LIN {X 0,Y 298.481,Z 502.932,A -85,B 0,C 180,E1 -16460.513,E2 -16460.513} C_VEL
LIN {X 0,Y 297.98,Z 506.123,A -85,B 0,C 180,E1 -16462.135,E2 -16462.135} C_VEL
LIN {X 0,Y 297.332,Z 509.748,A -85,B 0,C 180,E1 -16464.575,E2 -16464.575} C_VEL
LIN {X 0,Y 297.148,Z 511.131,A -85,B 0,C 180,E1 -16465.931,E2 -16465.931} C_VEL
LIN {X 0,Y 297.066,Z 512.111,A -85,B 0,C 180,E1 -16467.288,E2 -16467.288} C_VEL
LIN {X 0,Y 296.924,Z 512.947,A -85,B 0,C 180,E1 -16470,E2 -16470} C_VEL
LIN {X 0,Y 297.047,Z 512.175,A -85,B 0,C 180,E1 -16472.712,E2 -16472.712} C_VEL
LIN {X 0,Y 297.329,Z 509.873,A -85,B 0,C 180,E1 -16475.426,E2 -16475.426} C_VEL
LIN {X 0,Y 297.887,Z 506.563,A -85,B 0,C 180,E1 -16477.733,E2 -16477.733} C_VEL
LIN {X 0,Y 298.7,Z 501.616,A -85,B 0,C 180,E1 -16480.164,E2 -16480.164} C_VEL
LIN {X 0,Y 299.966,Z 495.208,A -85,B 0,C 180,E1 -16482.517,E2 -16482.517} C_VEL
LIN {X 0,Y 301.198,Z 488.167,A -85,B 0,C 180,E1 -16484.527,E2 -16484.527} C_VEL
LIN {X 0,Y 302.803,Z 479.382,A -85,B 0,C 180,E1 -16486.518,E2 -16486.518} C_VEL
LIN {X 0,Y 304.304,Z 470.362,A -85,B 0,C 180,E1 -16488.167,E2 -16488.167} C_VEL
LIN {X 0,Y 305.67,Z 460.096,A -85,B 0,C 180,E1 -16489.687,E2 -16489.687} C_VEL
LIN {X 0,Y 307.036,Z 449.246,A -85,B 0,C 180,E1 -16490.956,E2 -16490.956} C_VEL
LIN {X 0,Y 307.418,Z 446.051,A -85,B 0,C 180,E1 -16491.28,E2 -16491.28} C_VEL
LIN {X 0,Y 305.864,Z 437.325,A -85,B 0,C 180,E1 -16492.242,E2 -16492.242} C_VEL
LIN {X 0,Y 302.839,Z 425.594,A -85,B 0,C 180,E1 -16493.382,E2 -16493.382} C_VEL
LIN {X 0,Y 298.696,Z 412.913,A -85,B 0,C 180,E1 -16494.408,E2 -16494.408} C_VEL
LIN {X 0,Y 297.744,Z 409.886,A -85,B 0,C 180,E1 -16494.623,E2 -16494.623} C_VEL
LIN {X 0,Y 297.824,Z 406.969,A -85,B 0,C 180,E1 -16498.162,E2 -16498.162} C_VEL
LIN {X 0,Y 297.994,Z 404.067,A -85,B 0,C 180,E1 -16501.892,E2 -16501.892} C_VEL
LIN {X 0,Y 298.002,Z 403.367,A -85,B 0,C 180,E1 -16502.849,E2 -16502.849} C_VEL
LIN {X 0,Y 298.372,Z 403.32,A -85,B 0,C 180,E1 -16506.788,E2 -16506.788} C_VEL
LIN {X 0,Y 298.401,Z 403.313,A -85,B 0,C 180,E1 -16509.488,E2 -16509.488} C_VEL
LIN {X 0,Y 298.401,Z 403.313,A -85,B 0,C 180,E1 -16513.103,E2 -16513.103} C_VEL
LIN {X 0,Y 298.405,Z 403.313,A -85,B 0,C 180,E1 -16516.921,E2 -16516.921} C_VEL
LIN {X 0,Y 298.418,Z 403.309,A -85,B 0,C 180,E1 -16521.004,E2 -16521.004} C_VEL
LIN {X 0,Y 298.436,Z 403.311,A -85,B 0,C 180,E1 -16523.932,E2 -16523.932} C_VEL
LIN {X 0,Y 298.398,Z 403.316,A -85,B 0,C 180,E1 -16527.984,E2 -16527.984} C_VEL
LIN {X 0,Y 298.462,Z 403.308,A -85,B 0,C 180,E1 -16531.904,E2 -16531.904} C_VEL
LIN {X 0,Y 298.487,Z 403.301,A -85,B 0,C 180,E1 -16534.924,E2 -16534.924} C_VEL
LIN {X 0,Y 298.444,Z 403.308,A -85,B 0,C 180,E1 -16539.315,E2 -16539.315} C_VEL
LIN {X 0,Y 298.541,Z 403.298,A -85,B 0,C 180,E1 -16542.179,E2 -16542.179} C_VEL
LIN {X 0,Y 298.597,Z 403.288,A -85,B 0,C 180,E1 -16544.995,E2 -16544.995} C_VEL
LIN {X 0,Y 298.595,Z 403.288,A -85,B 0,C 180,E1 -16549.147,E2 -16549.147} C_VEL
LIN {X 0,Y 298.659,Z 403.281,A -85,B 0,C 180,E1 -16550.741,E2 -16550.741} C_VEL
LIN {X 0,Y 298.057,Z 403.359,A -85,B 0,C 180,E1 -16551.868,E2 -16551.868} C_VEL
LIN {X 0,Y 295.127,Z 403.725,A -85,B 0,C 180,E1 -16553.699,E2 -16553.699} C_VEL
LIN {X 0,Y 292.661,Z 404.03,A -85,B 0,C 180,E1 -16555.186,E2 -16555.186} C_VEL
LIN {X 0,Y 291.704,Z 404.15,A -85,B 0,C 180,E1 -16556.341,E2 -16556.341} C_VEL
LIN {X 0,Y 291.685,Z 404.15,A -85,B 0,C 180,E1 -16556.731,E2 -16556.731} C_VEL
LIN {X 0,Y 291.969,Z 404.118,A -85,B 0,C 180,E1 -16560,E2 -16560} C_VEL
LIN {X 0,Y 291.793,Z 404.138,A -85,B 0,C 180,E1 -16562.761,E2 -16562.761} C_VEL
LIN {X 0,Y 291.751,Z 404.142,A -85,B 0,C 180,E1 -16566.918,E2 -16566.918} C_VEL
LIN {X 0,Y 291.634,Z 404.16,A -85,B 0,C 180,E1 -16569.712,E2 -16569.712} C_VEL
LIN {X 0,Y 291.527,Z 404.17,A -85,B 0,C 180,E1 -16573.95,E2 -16573.95} C_VEL
LIN {X 0,Y 291.491,Z 404.173,A -85,B 0,C 180,E1 -16576.818,E2 -16576.818} C_VEL
LIN {X 0,Y 291.454,Z 404.179,A -85,B 0,C 180,E1 -16579.875,E2 -16579.875} C_VEL
LIN {X 0,Y 291.404,Z 404.185,A -85,B 0,C 180,E1 -16584.205,E2 -16584.205} C_VEL
LIN {X 0,Y 291.423,Z 404.186,A -85,B 0,C 180,E1 -16587.272,E2 -16587.272} C_VEL
LIN {X 0,Y 291.337,Z 404.195,A -85,B 0,C 180,E1 -16590.437,E2 -16590.437} C_VEL
LIN {X 0,Y 291.348,Z 404.195,A -85,B 0,C 180,E1 -16593.698,E2 -16593.698} C_VEL
LIN {X 0,Y 291.379,Z 404.189,A -85,B 0,C 180,E1 -16597.254,E2 -16597.254} C_VEL
LIN {X 0,Y 291.384,Z 404.329,A -85,B 0,C 180,E1 -16598.622,E2 -16598.622} C_VEL
LIN {X 0,Y 292.173,Z 408.492,A -85,B 0,C 180,E1 -16602.339,E2 -16602.339} C_VEL
LIN {X 0,Y 292.99,Z 412.972,A -85,B 0,C 180,E1 -16606.023,E2 -16606.023} C_VEL
LIN {X 0,Y 293.883,Z 418.089,A -85,B 0,C 180,E1 -16609.93,E2 -16609.93} C_VEL
LIN {X 0,Y 294.289,Z 420.975,A -85,B 0,C 180,E1 -16612.007,E2 -16612.007} C_VEL
LIN {X 0,Y 294.149,Z 424.38,A -85,B 0,C 180,E1 -16614.326,E2 -16614.326} C_VEL
LIN {X 0,Y 293.105,Z 430.281,A -85,B 0,C 180,E1 -16618.162,E2 -16618.162} C_VEL
LIN {X 0,Y 292.109,Z 436.327,A -85,B 0,C 180,E1 -16622.02,E2 -16622.02} C_VEL
LIN {X 0,Y 291.475,Z 440.717,A -85,B 0,C 180,E1 -16624.804,E2 -16624.804} C_VEL
LIN {X 0,Y 294.39,Z 454.459,A -85,B 0,C 180,E1 -16625.683,E2 -16625.683} C_VEL
LIN {X 0,Y 296.244,Z 466.513,A -85,B 0,C 180,E1 -16626.656,E2 -16626.656} C_VEL
LIN {X 0,Y 297.356,Z 478.025,A -85,B 0,C 180,E1 -16627.78,E2 -16627.78} C_VEL
LIN {X 0,Y 297.893,Z 489.194,A -85,B 0,C 180,E1 -16629.094,E2 -16629.094} C_VEL
LIN {X 0,Y 297.365,Z 494.548,A -85,B 0,C 180,E1 -16629.778,E2 -16629.778} C_VEL
LIN {X 0,Y 295.651,Z 504.76,A -85,B 0,C 180,E1 -16631.282,E2 -16631.282} C_VEL
LIN {X 0,Y 294.109,Z 514.527,A -85,B 0,C 180,E1 -16633.099,E2 -16633.099} C_VEL
LIN {X 0,Y 292.637,Z 522.957,A -85,B 0,C 180,E1 -16635.038,E2 -16635.038} C_VEL
LIN {X 0,Y 291.387,Z 530.195,A -85,B 0,C 180,E1 -16637.108,E2 -16637.108} C_VEL
LIN {X 0,Y 290.676,Z 535.094,A -85,B 0,C 180,E1 -16638.847,E2 -16638.847} C_VEL
LIN {X 0,Y 290.06,Z 539.861,A -85,B 0,C 180,E1 -16640.938,E2 -16640.938} C_VEL
LIN {X 0,Y 289.753,Z 543.515,A -85,B 0,C 180,E1 -16643.034,E2 -16643.034} C_VEL
LIN {X 0,Y 289.625,Z 545.401,A -85,B 0,C 180,E1 -16644.43,E2 -16644.43} C_VEL
LIN {X 0,Y 289.583,Z 546.818,A -85,B 0,C 180,E1 -16645.825,E2 -16645.825} C_VEL
LIN {X 0,Y 289.563,Z 547.831,A -85,B 0,C 180,E1 -16647.217,E2 -16647.217} C_VEL
LIN {X 0,Y 289.586,Z 548.45,A -85,B 0,C 180,E1 -16648.609,E2 -16648.609} C_VEL
LIN {X 0,Y 289.693,Z 548.674,A -85,B 0,C 180,E1 -16650,E2 -16650} C_VEL
LIN {X 0,Y 289.606,Z 548.447,A -85,B 0,C 180,E1 -16651.39,E2 -16651.39} C_VEL
LIN {X 0,Y 289.563,Z 547.824,A -85,B 0,C 180,E1 -16652.782,E2 -16652.782} C_VEL
LIN {X 0,Y 289.582,Z 546.81,A -85,B 0,C 180,E1 -16654.175,E2 -16654.175} C_VEL
LIN {X 0,Y 289.632,Z 545.091,A -85,B 0,C 180,E1 -16655.802,E2 -16655.802} C_VEL
LIN {X 0,Y 289.906,Z 541.16,A -85,B 0,C 180,E1 -16658.363,E2 -16658.363} C_VEL
LIN {X 0,Y 290.449,Z 536.77,A -85,B 0,C 180,E1 -16660.456,E2 -16660.456} C_VEL
LIN {X 0,Y 291.198,Z 531.183,A -85,B 0,C 180,E1 -16662.545,E2 -16662.545} C_VEL
LIN {X 0,Y 292.458,Z 524.234,A -85,B 0,C 180,E1 -16664.615,E2 -16664.615} C_VEL
LIN {X 0,Y 293.956,Z 515.544,A -85,B 0,C 180,E1 -16666.672,E2 -16666.672} C_VEL
LIN {X 0,Y 295.281,Z 506.633,A -85,B 0,C 180,E1 -16668.383,E2 -16668.383} C_VEL
LIN {X 0,Y 297.128,Z 495.697,A -85,B 0,C 180,E1 -16670.058,E2 -16670.058} C_VEL
LIN {X 0,Y 297.903,Z 490.505,A -85,B 0,C 180,E1 -16670.724,E2 -16670.724} C_VEL
LIN {X 0,Y 297.452,Z 479.648,A -85,B 0,C 180,E1 -16672.029,E2 -16672.029} C_VEL
LIN {X 0,Y 296.313,Z 467.11,A -85,B 0,C 180,E1 -16673.271,E2 -16673.271} C_VEL
LIN {X 0,Y 294.317,Z 453.871,A -85,B 0,C 180,E1 -16674.337,E2 -16674.337} C_VEL
LIN {X 0,Y 291.471,Z 440.636,A -85,B 0,C 180,E1 -16675.196,E2 -16675.196} C_VEL
LIN {X 0,Y 292.495,Z 433.977,A -85,B 0,C 180,E1 -16679.454,E2 -16679.454} C_VEL
LIN {X 0,Y 293.547,Z 427.802,A -85,B 0,C 180,E1 -16683.412,E2 -16683.412} C_VEL
LIN {X 0,Y 294.37,Z 422.88,A -85,B 0,C 180,E1 -16686.646,E2 -16686.646} C_VEL
LIN {X 0,Y 294.101,Z 419.178,A -85,B 0,C 180,E1 -16689.218,E2 -16689.218} C_VEL
LIN {X 0,Y 293.195,Z 414.034,A -85,B 0,C 180,E1 -16693.054,E2 -16693.054} C_VEL
LIN {X 0,Y 292.447,Z 410.214,A -85,B 0,C 180,E1 -16696.133,E2 -16696.133} C_VEL
LIN {X 0,Y 291.757,Z 406.402,A -85,B 0,C 180,E1 -16699.429,E2 -16699.429} C_VEL
LIN {X 0,Y 291.362,Z 404.194,A -85,B 0,C 180,E1 -16701.588,E2 -16701.588} C_VEL
LIN {X 0,Y 291.371,Z 404.194,A -85,B 0,C 180,E1 -16705.095,E2 -16705.095} C_VEL
LIN {X 0,Y 291.373,Z 404.191,A -85,B 0,C 180,E1 -16707.951,E2 -16707.951} C_VEL
LIN {X 0,Y 291.38,Z 404.19,A -85,B 0,C 180,E1 -16711.158,E2 -16711.158} C_VEL
LIN {X 0,Y 291.416,Z 404.185,A -85,B 0,C 180,E1 -16714.272,E2 -16714.272} C_VEL
LIN {X 0,Y 291.384,Z 404.188,A -85,B 0,C 180,E1 -16717.3,E2 -16717.3} C_VEL
LIN {X 0,Y 291.46,Z 404.18,A -85,B 0,C 180,E1 -16720.27,E2 -16720.27} C_VEL
LIN {X 0,Y 291.557,Z 404.169,A -85,B 0,C 180,E1 -16724.624,E2 -16724.624} C_VEL
LIN {X 0,Y 291.541,Z 404.17,A -85,B 0,C 180,E1 -16728.881,E2 -16728.881} C_VEL
LIN {X 0,Y 291.712,Z 404.147,A -85,B 0,C 180,E1 -16731.689,E2 -16731.689} C_VEL
LIN {X 0,Y 291.633,Z 404.16,A -85,B 0,C 180,E1 -16734.468,E2 -16734.468} C_VEL
LIN {X 0,Y 291.893,Z 404.126,A -85,B 0,C 180,E1 -16738.62,E2 -16738.62} C_VEL
LIN {X 0,Y 291.892,Z 404.123,A -85,B 0,C 180,E1 -16741.38,E2 -16741.38} C_VEL
LIN {X 0,Y 291.75,Z 404.141,A -85,B 0,C 180,E1 -16746.918,E2 -16746.918} C_VEL
LIN {X 0,Y 291.632,Z 404.157,A -85,B 0,C 180,E1 -16749.712,E2 -16749.712} C_VEL
LIN {X 0,Y 291.525,Z 404.172,A -85,B 0,C 180,E1 -16753.95,E2 -16753.95} C_VEL
LIN {X 0,Y 291.489,Z 404.174,A -85,B 0,C 180,E1 -16756.818,E2 -16756.818} C_VEL
LIN {X 0,Y 291.453,Z 404.181,A -85,B 0,C 180,E1 -16759.875,E2 -16759.875} C_VEL
LIN {X 0,Y 291.385,Z 404.189,A -85,B 0,C 180,E1 -16764.207,E2 -16764.207} C_VEL
LIN {X 0,Y 291.422,Z 404.182,A -85,B 0,C 180,E1 -16767.272,E2 -16767.272} C_VEL
LIN {X 0,Y 291.336,Z 404.194,A -85,B 0,C 180,E1 -16770.437,E2 -16770.437} C_VEL
LIN {X 0,Y 291.347,Z 404.192,A -85,B 0,C 180,E1 -16773.698,E2 -16773.698} C_VEL
LIN {X 0,Y 291.396,Z 404.184,A -85,B 0,C 180,E1 -16777.259,E2 -16777.259} C_VEL
LIN {X 0,Y 291.337,Z 404.192,A -85,B 0,C 180,E1 -16780.642,E2 -16780.642} C_VEL
LIN {X 0,Y 291.344,Z 404.192,A -85,B 0,C 180,E1 -16784.392,E2 -16784.392} C_VEL
LIN {X 0,Y 291.389,Z 404.188,A -85,B 0,C 180,E1 -16788.391,E2 -16788.391} C_VEL
LIN {X 0,Y 291.366,Z 404.193,A -85,B 0,C 180,E1 -16791.16,E2 -16791.16} C_VEL
LIN {X 0,Y 291.181,Z 404.217,A -85,B 0,C 180,E1 -16794.601,E2 -16794.601} C_VEL
LIN {X 0,Y 291.028,Z 404.237,A -85,B 0,C 180,E1 -16796.26,E2 -16796.26} C_VEL
LIN {X 0,Y 290.946,Z 404.865,A -85,B 0,C 180,E1 -16797.898,E2 -16797.898} C_VEL
LIN {X 0,Y 290.821,Z 407.307,A -85,B 0,C 180,E1 -16801.097,E2 -16801.097} C_VEL
LIN {X 0,Y 290.717,Z 410.398,A -85,B 0,C 180,E1 -16804.867,E2 -16804.867} C_VEL
LIN {X 0,Y 295.063,Z 423.319,A -85,B 0,C 180,E1 -16805.909,E2 -16805.909} C_VEL
LIN {X 0,Y 298.513,Z 435.452,A -85,B 0,C 180,E1 -16807.093,E2 -16807.093} C_VEL
LIN {X 0,Y 300.478,Z 445.399,A -85,B 0,C 180,E1 -16808.204,E2 -16808.204} C_VEL
LIN {X 0,Y 300.584,Z 448.677,A -85,B 0,C 180,E1 -16808.572,E2 -16808.572} C_VEL
LIN {X 0,Y 299.092,Z 459.652,A -85,B 0,C 180,E1 -16809.853,E2 -16809.853} C_VEL
LIN {X 0,Y 297.608,Z 470.166,A -85,B 0,C 180,E1 -16811.41,E2 -16811.41} C_VEL
LIN {X 0,Y 296.07,Z 479.299,A -85,B 0,C 180,E1 -16813.095,E2 -16813.095} C_VEL
LIN {X 0,Y 294.636,Z 486.829,A -85,B 0,C 180,E1 -16814.788,E2 -16814.788} C_VEL
LIN {X 0,Y 293.324,Z 494.192,A -85,B 0,C 180,E1 -16816.843,E2 -16816.843} C_VEL
LIN {X 0,Y 292.087,Z 500.107,A -85,B 0,C 180,E1 -16818.902,E2 -16818.902} C_VEL
LIN {X 0,Y 291.288,Z 504.768,A -85,B 0,C 180,E1 -16820.977,E2 -16820.977} C_VEL
LIN {X 0,Y 290.641,Z 508.336,A -85,B 0,C 180,E1 -16823.056,E2 -16823.056} C_VEL
LIN {X 0,Y 290.292,Z 510.18,A -85,B 0,C 180,E1 -16824.443,E2 -16824.443} C_VEL
LIN {X 0,Y 290.078,Z 511.563,A -85,B 0,C 180,E1 -16825.832,E2 -16825.832} C_VEL
LIN {X 0,Y 289.983,Z 512.544,A -85,B 0,C 180,E1 -16827.222,E2 -16827.222} C_VEL
LIN {X 0,Y 289.838,Z 513.379,A -85,B 0,C 180,E1 -16830,E2 -16830} C_VEL
LIN {X 0,Y 289.858,Z 513.188,A -85,B 0,C 180,E1 -16831.389,E2 -16831.389} C_VEL
LIN {X 0,Y 289.964,Z 512.606,A -85,B 0,C 180,E1 -16832.779,E2 -16832.779} C_VEL
LIN {X 0,Y 290.29,Z 510.303,A -85,B 0,C 180,E1 -16835.557,E2 -16835.557} C_VEL
LIN {X 0,Y 290.851,Z 507.177,A -85,B 0,C 180,E1 -16837.815,E2 -16837.815} C_VEL
LIN {X 0,Y 291.444,Z 503.595,A -85,B 0,C 180,E1 -16839.718,E2 -16839.718} C_VEL
LIN {X 0,Y 292.434,Z 498.605,A -85,B 0,C 180,E1 -16841.787,E2 -16841.787} C_VEL
LIN {X 0,Y 293.667,Z 492.316,A -85,B 0,C 180,E1 -16843.847,E2 -16843.847} C_VEL
LIN {X 0,Y 295.118,Z 484.444,A -85,B 0,C 180,E1 -16845.895,E2 -16845.895} C_VEL
LIN {X 0,Y 296.652,Z 476.406,A -85,B 0,C 180,E1 -16847.582,E2 -16847.582} C_VEL
LIN {X 0,Y 298.184,Z 466.603,A -85,B 0,C 180,E1 -16849.267,E2 -16849.267} C_VEL
LIN {X 0,Y 299.495,Z 456.948,A -85,B 0,C 180,E1 -16850.609,E2 -16850.609} C_VEL
LIN {X 0,Y 300.693,Z 446.485,A -85,B 0,C 180,E1 -16851.78,E2 -16851.78} C_VEL
LIN {X 0,Y 298.439,Z 435.44,A -85,B 0,C 180,E1 -16853.03,E2 -16853.03} C_VEL
LIN {X 0,Y 295.032,Z 423.054,A -85,B 0,C 180,E1 -16854.227,E2 -16854.227} C_VEL
LIN {X 0,Y 290.697,Z 410.312,A -85,B 0,C 180,E1 -16855.287,E2 -16855.287} C_VEL
LIN {X 0,Y 290.884,Z 406.875,A -85,B 0,C 180,E1 -16859.565,E2 -16859.565} C_VEL
LIN {X 0,Y 290.965,Z 404.835,A -85,B 0,C 180,E1 -16862.285,E2 -16862.285} C_VEL
LIN {X 0,Y 291.034,Z 404.235,A -85,B 0,C 180,E1 -16863.74,E2 -16863.74} C_VEL
LIN {X 0,Y 291.32,Z 404.197,A -85,B 0,C 180,E1 -16867.239,E2 -16867.239} C_VEL
LIN {X 0,Y 291.334,Z 404.196,A -85,B 0,C 180,E1 -16870.643,E2 -16870.643} C_VEL
LIN {X 0,Y 291.293,Z 404.202,A -85,B 0,C 180,E1 -16874.402,E2 -16874.402} C_VEL
LIN {X 0,Y 291.329,Z 404.196,A -85,B 0,C 180,E1 -16878.404,E2 -16878.404} C_VEL
LIN {X 0,Y 291.368,Z 404.187,A -85,B 0,C 180,E1 -16881.16,E2 -16881.16} C_VEL
LIN {X 0,Y 291.389,Z 404.187,A -85,B 0,C 180,E1 -16884.63,E2 -16884.63} C_VEL
LIN {X 0,Y 291.375,Z 404.191,A -85,B 0,C 180,E1 -16887.951,E2 -16887.951} C_VEL
LIN {X 0,Y 291.381,Z 404.187,A -85,B 0,C 180,E1 -16891.158,E2 -16891.158} C_VEL
LIN {X 0,Y 291.417,Z 404.185,A -85,B 0,C 180,E1 -16894.272,E2 -16894.272} C_VEL
LIN {X 0,Y 291.378,Z 404.188,A -85,B 0,C 180,E1 -16897.299,E2 -16897.299} C_VEL
LIN {X 0,Y 291.461,Z 404.179,A -85,B 0,C 180,E1 -16900.27,E2 -16900.27} C_VEL
LIN {X 0,Y 291.559,Z 404.165,A -85,B 0,C 180,E1 -16904.624,E2 -16904.624} C_VEL
LIN {X 0,Y 291.539,Z 404.167,A -85,B 0,C 180,E1 -16908.881,E2 -16908.881} C_VEL
LIN {X 0,Y 291.672,Z 404.155,A -85,B 0,C 180,E1 -16911.687,E2 -16911.687} C_VEL
LIN {X 0,Y 291.628,Z 404.157,A -85,B 0,C 180,E1 -16914.468,E2 -16914.468} C_VEL
LIN {X 0,Y 291.685,Z 404.15,A -85,B 0,C 180,E1 -16916.731,E2 -16916.731} C_VEL
LIN {X 0,Y 291.215,Z 404.212,A -85,B 0,C 180,E1 -16917.885,E2 -16917.885} C_VEL
LIN {X 0,Y 289.773,Z 404.394,A -85,B 0,C 180,E1 -16919.02,E2 -16919.02} C_VEL
LIN {X 0,Y 285.193,Z 404.965,A -85,B 0,C 180,E1 -16922.078,E2 -16922.078} C_VEL
LIN {X 0,Y 284.736,Z 405.017,A -85,B 0,C 180,E1 -16922.877,E2 -16922.877} C_VEL
LIN {X 0,Y 284.703,Z 405.021,A -85,B 0,C 180,E1 -16927.09,E2 -16927.09} C_VEL
LIN {X 0,Y 284.571,Z 405.038,A -85,B 0,C 180,E1 -16929.955,E2 -16929.955} C_VEL
LIN {X 0,Y 284.487,Z 405.046,A -85,B 0,C 180,E1 -16934.303,E2 -16934.303} C_VEL
LIN {X 0,Y 284.429,Z 405.053,A -85,B 0,C 180,E1 -16937.248,E2 -16937.248} C_VEL
LIN {X 0,Y 284.382,Z 405.058,A -85,B 0,C 180,E1 -16940.242,E2 -16940.242} C_VEL
LIN {X 0,Y 284.373,Z 405.062,A -85,B 0,C 180,E1 -16943.875,E2 -16943.875} C_VEL
LIN {X 0,Y 284.398,Z 405.061,A -85,B 0,C 180,E1 -16947.173,E2 -16947.173} C_VEL
LIN {X 0,Y 284.297,Z 405.074,A -85,B 0,C 180,E1 -16951.274,E2 -16951.274} C_VEL
LIN {X 0,Y 284.344,Z 405.064,A -85,B 0,C 180,E1 -16955.348,E2 -16955.348} C_VEL
LIN {X 0,Y 284.343,Z 405.102,A -85,B 0,C 180,E1 -16957.882,E2 -16957.882} C_VEL
LIN {X 0,Y 285.24,Z 409.942,A -85,B 0,C 180,E1 -16962.339,E2 -16962.339} C_VEL
LIN {X 0,Y 286.158,Z 414.973,A -85,B 0,C 180,E1 -16966.553,E2 -16966.553} C_VEL
LIN {X 0,Y 287.026,Z 420.007,A -85,B 0,C 180,E1 -16970.459,E2 -16970.459} C_VEL
LIN {X 0,Y 287.315,Z 423.728,A -85,B 0,C 180,E1 -16973.159,E2 -16973.159} C_VEL
LIN {X 0,Y 286.494,Z 428.687,A -85,B 0,C 180,E1 -16976.518,E2 -16976.518} C_VEL
LIN {X 0,Y 285.428,Z 434.704,A -85,B 0,C 180,E1 -16980.498,E2 -16980.498} C_VEL
LIN {X 0,Y 284.544,Z 440.291,A -85,B 0,C 180,E1 -16984.153,E2 -16984.153} C_VEL
LIN {X 0,Y 287.442,Z 453.667,A -85,B 0,C 180,E1 -16985.035,E2 -16985.035} C_VEL
LIN {X 0,Y 289.48,Z 466.517,A -85,B 0,C 180,E1 -16986.114,E2 -16986.114} C_VEL
LIN {X 0,Y 290.598,Z 478.93,A -85,B 0,C 180,E1 -16987.376,E2 -16987.376} C_VEL
LIN {X 0,Y 291.073,Z 490.191,A -85,B 0,C 180,E1 -16988.766,E2 -16988.766} C_VEL
LIN {X 0,Y 290.264,Z 496.56,A -85,B 0,C 180,E1 -16989.631,E2 -16989.631} C_VEL
LIN {X 0,Y 288.536,Z 506.292,A -85,B 0,C 180,E1 -16991.171,E2 -16991.171} C_VEL
LIN {X 0,Y 287.089,Z 515.183,A -85,B 0,C 180,E1 -16992.916,E2 -16992.916} C_VEL
LIN {X 0,Y 285.533,Z 523.855,A -85,B 0,C 180,E1 -16995.022,E2 -16995.022} C_VEL
LIN {X 0,Y 284.238,Z 530.793,A -85,B 0,C 180,E1 -16997.142,E2 -16997.142} C_VEL
LIN {X 0,Y 283.427,Z 536.372,A -85,B 0,C 180,E1 -16999.282,E2 -16999.282} C_VEL
LIN {X 0,Y 282.877,Z 540.755,A -85,B 0,C 180,E1 -17001.427,E2 -17001.427} C_VEL
LIN {X 0,Y 282.681,Z 543.081,A -85,B 0,C 180,E1 -17002.859,E2 -17002.859} C_VEL
LIN {X 0,Y 282.563,Z 544.969,A -85,B 0,C 180,E1 -17004.29,E2 -17004.29} C_VEL
LIN {X 0,Y 282.503,Z 546.386,A -85,B 0,C 180,E1 -17005.72,E2 -17005.72} C_VEL
LIN {X 0,Y 282.489,Z 547.4,A -85,B 0,C 180,E1 -17007.148,E2 -17007.148} C_VEL
LIN {X 0,Y 282.5,Z 548.019,A -85,B 0,C 180,E1 -17008.574,E2 -17008.574} C_VEL
LIN {X 0,Y 282.604,Z 548.243,A -85,B 0,C 180,E1 -17010,E2 -17010} C_VEL
LIN {X 0,Y 282.519,Z 548.015,A -85,B 0,C 180,E1 -17011.425,E2 -17011.425} C_VEL
LIN {X 0,Y 282.489,Z 547.393,A -85,B 0,C 180,E1 -17012.852,E2 -17012.852} C_VEL
LIN {X 0,Y 282.502,Z 546.377,A -85,B 0,C 180,E1 -17014.28,E2 -17014.28} C_VEL
LIN {X 0,Y 282.558,Z 544.868,A -85,B 0,C 180,E1 -17015.782,E2 -17015.782} C_VEL
LIN {X 0,Y 282.74,Z 541.97,A -85,B 0,C 180,E1 -17017.858,E2 -17017.858} C_VEL
LIN {X 0,Y 283.195,Z 537.944,A -85,B 0,C 180,E1 -17020.004,E2 -17020.004} C_VEL
LIN {X 0,Y 284.074,Z 531.767,A -85,B 0,C 180,E1 -17022.502,E2 -17022.502} C_VEL
LIN {X 0,Y 285.333,Z 525.043,A -85,B 0,C 180,E1 -17024.623,E2 -17024.623} C_VEL
LIN {X 0,Y 286.847,Z 516.706,A -85,B 0,C 180,E1 -17026.731,E2 -17026.731} C_VEL
LIN {X 0,Y 288.189,Z 508.156,A -85,B 0,C 180,E1 -17028.483,E2 -17028.483} C_VEL
LIN {X 0,Y 290.044,Z 497.622,A -85,B 0,C 180,E1 -17030.199,E2 -17030.199} C_VEL
LIN {X 0,Y 291.064,Z 491.392,A -85,B 0,C 180,E1 -17031.049,E2 -17031.049} C_VEL
LIN {X 0,Y 290.646,Z 480.023,A -85,B 0,C 180,E1 -17032.486,E2 -17032.486} C_VEL
LIN {X 0,Y 289.572,Z 467.646,A -85,B 0,C 180,E1 -17033.763,E2 -17033.763} C_VEL
LIN {X 0,Y 287.664,Z 454.808,A -85,B 0,C 180,E1 -17034.852,E2 -17034.852} C_VEL
LIN {X 0,Y 284.689,Z 441.541,A -85,B 0,C 180,E1 -17035.77,E2 -17035.77} C_VEL
LIN {X 0,Y 284.522,Z 440.174,A -85,B 0,C 180,E1 -17035.863,E2 -17035.863} C_VEL
LIN {X 0,Y 285.423,Z 434.665,A -85,B 0,C 180,E1 -17039.503,E2 -17039.503} C_VEL
LIN {X 0,Y 286.5,Z 428.643,A -85,B 0,C 180,E1 -17043.484,E2 -17043.484} C_VEL
LIN {X 0,Y 287.348,Z 423.673,A -85,B 0,C 180,E1 -17046.841,E2 -17046.841} C_VEL
LIN {X 0,Y 287.027,Z 419.951,A -85,B 0,C 180,E1 -17049.541,E2 -17049.541} C_VEL
LIN {X 0,Y 286.137,Z 414.877,A -85,B 0,C 180,E1 -17053.45,E2 -17053.45} C_VEL
LIN {X 0,Y 285.168,Z 409.864,A -85,B 0,C 180,E1 -17057.677,E2 -17057.677} C_VEL
LIN {X 0,Y 284.376,Z 405.353,A -85,B 0,C 180,E1 -17061.841,E2 -17061.841} C_VEL
LIN {X 0,Y 284.337,Z 405.066,A -85,B 0,C 180,E1 -17062.274,E2 -17062.274} C_VEL
LIN {X 0,Y 284.31,Z 405.073,A -85,B 0,C 180,E1 -17065.351,E2 -17065.351} C_VEL
LIN {X 0,Y 284.296,Z 405.071,A -85,B 0,C 180,E1 -17068.726,E2 -17068.726} C_VEL
LIN {X 0,Y 284.397,Z 405.061,A -85,B 0,C 180,E1 -17072.827,E2 -17072.827} C_VEL
LIN {X 0,Y 284.369,Z 405.065,A -85,B 0,C 180,E1 -17076.707,E2 -17076.707} C_VEL
LIN {X 0,Y 284.406,Z 405.057,A -85,B 0,C 180,E1 -17081.262,E2 -17081.262} C_VEL
LIN {X 0,Y 284.494,Z 405.05,A -85,B 0,C 180,E1 -17084.459,E2 -17084.459} C_VEL
LIN {X 0,Y 284.493,Z 405.05,A -85,B 0,C 180,E1 -17088.602,E2 -17088.602} C_VEL
LIN {X 0,Y 284.662,Z 405.025,A -85,B 0,C 180,E1 -17091.481,E2 -17091.481} C_VEL
LIN {X 0,Y 284.604,Z 405.035,A -85,B 0,C 180,E1 -17094.331,E2 -17094.331} C_VEL
LIN {X 0,Y 284.858,Z 405.002,A -85,B 0,C 180,E1 -17098.586,E2 -17098.586} C_VEL
LIN {X 0,Y 284.858,Z 404.999,A -85,B 0,C 180,E1 -17101.414,E2 -17101.414} C_VEL
LIN {X 0,Y 284.702,Z 405.018,A -85,B 0,C 180,E1 -17107.09,E2 -17107.09} C_VEL
LIN {X 0,Y 284.569,Z 405.038,A -85,B 0,C 180,E1 -17109.955,E2 -17109.955} C_VEL
LIN {X 0,Y 284.484,Z 405.05,A -85,B 0,C 180,E1 -17114.303,E2 -17114.303} C_VEL
LIN {X 0,Y 284.428,Z 405.053,A -85,B 0,C 180,E1 -17117.248,E2 -17117.248} C_VEL
LIN {X 0,Y 284.38,Z 405.062,A -85,B 0,C 180,E1 -17120.242,E2 -17120.242} C_VEL
LIN {X 0,Y 284.34,Z 405.064,A -85,B 0,C 180,E1 -17124.847,E2 -17124.847} C_VEL
LIN {X 0,Y 284.331,Z 405.07,A -85,B 0,C 180,E1 -17128.011,E2 -17128.011} C_VEL
LIN {X 0,Y 284.296,Z 405.071,A -85,B 0,C 180,E1 -17131.274,E2 -17131.274} C_VEL
LIN {X 0,Y 284.364,Z 405.063,A -85,B 0,C 180,E1 -17135.354,E2 -17135.354} C_VEL
LIN {X 0,Y 284.325,Z 405.068,A -85,B 0,C 180,E1 -17138.167,E2 -17138.167} C_VEL
LIN {X 0,Y 284.285,Z 405.072,A -85,B 0,C 180,E1 -17142.128,E2 -17142.128} C_VEL
LIN {X 0,Y 284.32,Z 405.069,A -85,B 0,C 180,E1 -17146.202,E2 -17146.202} C_VEL
LIN {X 0,Y 284.353,Z 405.067,A -85,B 0,C 180,E1 -17150.013,E2 -17150.013} C_VEL
LIN {X 0,Y 284.215,Z 405.087,A -85,B 0,C 180,E1 -17153.597,E2 -17153.597} C_VEL
LIN {X 0,Y 283.904,Z 405.307,A -85,B 0,C 180,E1 -17157.002,E2 -17157.002} C_VEL
LIN {X 0,Y 283.848,Z 407.739,A -85,B 0,C 180,E1 -17160.317,E2 -17160.317} C_VEL
LIN {X 0,Y 283.701,Z 410.829,A -85,B 0,C 180,E1 -17164.197,E2 -17164.197} C_VEL
LIN {X 0,Y 288.138,Z 423.724,A -85,B 0,C 180,E1 -17165.287,E2 -17165.287} C_VEL
LIN {X 0,Y 291.708,Z 436.323,A -85,B 0,C 180,E1 -17166.562,E2 -17166.562} C_VEL
LIN {X 0,Y 293.94,Z 447.553,A -85,B 0,C 180,E1 -17167.878,E2 -17167.878} C_VEL
LIN {X 0,Y 293.596,Z 452.251,A -85,B 0,C 180,E1 -17168.405,E2 -17168.405} C_VEL
LIN {X 0,Y 291.945,Z 463.55,A -85,B 0,C 180,E1 -17169.86,E2 -17169.86} C_VEL
LIN {X 0,Y 290.596,Z 472.547,A -85,B 0,C 180,E1 -17171.31,E2 -17171.31} C_VEL
LIN {X 0,Y 288.941,Z 481.349,A -85,B 0,C 180,E1 -17173.029,E2 -17173.029} C_VEL
LIN {X 0,Y 287.303,Z 489.925,A -85,B 0,C 180,E1 -17175.117,E2 -17175.117} C_VEL
LIN {X 0,Y 285.974,Z 496.753,A -85,B 0,C 180,E1 -17177.222,E2 -17177.222} C_VEL
LIN {X 0,Y 284.816,Z 502.221,A -85,B 0,C 180,E1 -17179.335,E2 -17179.335} C_VEL
LIN {X 0,Y 284.055,Z 506.502,A -85,B 0,C 180,E1 -17181.463,E2 -17181.463} C_VEL
LIN {X 0,Y 283.609,Z 508.768,A -85,B 0,C 180,E1 -17182.883,E2 -17182.883} C_VEL
LIN {X 0,Y 283.255,Z 510.611,A -85,B 0,C 180,E1 -17184.304,E2 -17184.304} C_VEL
LIN {X 0,Y 282.901,Z 512.976,A -85,B 0,C 180,E1 -17187.152,E2 -17187.152} C_VEL
LIN {X 0,Y 282.752,Z 513.811,A -85,B 0,C 180,E1 -17190,E2 -17190} C_VEL
LIN {X 0,Y 282.774,Z 513.62,A -85,B 0,C 180,E1 -17191.424,E2 -17191.424} C_VEL
LIN {X 0,Y 282.881,Z 513.038,A -85,B 0,C 180,E1 -17192.848,E2 -17192.848} C_VEL
LIN {X 0,Y 283.254,Z 510.733,A -85,B 0,C 180,E1 -17195.696,E2 -17195.696} C_VEL
LIN {X 0,Y 283.789,Z 507.837,A -85,B 0,C 180,E1 -17197.862,E2 -17197.862} C_VEL
LIN {X 0,Y 284.46,Z 504.026,A -85,B 0,C 180,E1 -17199.959,E2 -17199.959} C_VEL
LIN {X 0,Y 285.501,Z 499.035,A -85,B 0,C 180,E1 -17202.078,E2 -17202.078} C_VEL
LIN {X 0,Y 286.773,Z 492.747,A -85,B 0,C 180,E1 -17204.186,E2 -17204.186} C_VEL
LIN {X 0,Y 288.294,Z 484.874,A -85,B 0,C 180,E1 -17206.281,E2 -17206.281} C_VEL
LIN {X 0,Y 290.27,Z 475.063,A -85,B 0,C 180,E1 -17208.346,E2 -17208.346} C_VEL
LIN {X 0,Y 291.751,Z 465.032,A -85,B 0,C 180,E1 -17210.036,E2 -17210.036} C_VEL
LIN {X 0,Y 293.26,Z 454.569,A -85,B 0,C 180,E1 -17211.437,E2 -17211.437} C_VEL
LIN {X 0,Y 294.024,Z 448.526,A -85,B 0,C 180,E1 -17212.115,E2 -17212.115} C_VEL
LIN {X 0,Y 292.387,Z 439.401,A -85,B 0,C 180,E1 -17213.212,E2 -17213.212} C_VEL
LIN {X 0,Y 289.462,Z 427.969,A -85,B 0,C 180,E1 -17214.425,E2 -17214.425} C_VEL
LIN {X 0,Y 285.54,Z 416.154,A -85,B 0,C 180,E1 -17215.508,E2 -17215.508} C_VEL
LIN {X 0,Y 283.699,Z 410.783,A -85,B 0,C 180,E1 -17215.926,E2 -17215.926} C_VEL
LIN {X 0,Y 283.886,Z 407.625,A -85,B 0,C 180,E1 -17219.948,E2 -17219.948} C_VEL
LIN {X 0,Y 283.946,Z 405.395,A -85,B 0,C 180,E1 -17222.993,E2 -17222.993} C_VEL
LIN {X 0,Y 284.21,Z 405.085,A -85,B 0,C 180,E1 -17226.404,E2 -17226.404} C_VEL
LIN {X 0,Y 284.308,Z 405.07,A -85,B 0,C 180,E1 -17229.995,E2 -17229.995} C_VEL
LIN {X 0,Y 284.248,Z 405.079,A -85,B 0,C 180,E1 -17234.191,E2 -17234.191} C_VEL
LIN {X 0,Y 284.275,Z 405.074,A -85,B 0,C 180,E1 -17238.125,E2 -17238.125} C_VEL
LIN {X 0,Y 284.339,Z 405.068,A -85,B 0,C 180,E1 -17242.275,E2 -17242.275} C_VEL
LIN {X 0,Y 284.327,Z 405.064,A -85,B 0,C 180,E1 -17245.353,E2 -17245.353} C_VEL
LIN {X 0,Y 284.297,Z 405.071,A -85,B 0,C 180,E1 -17248.726,E2 -17248.726} C_VEL
LIN {X 0,Y 284.398,Z 405.057,A -85,B 0,C 180,E1 -17252.827,E2 -17252.827} C_VEL
LIN {X 0,Y 284.337,Z 405.065,A -85,B 0,C 180,E1 -17256.704,E2 -17256.704} C_VEL
LIN {X 0,Y 284.407,Z 405.056,A -85,B 0,C 180,E1 -17261.262,E2 -17261.262} C_VEL
LIN {X 0,Y 284.496,Z 405.046,A -85,B 0,C 180,E1 -17264.459,E2 -17264.459} C_VEL
LIN {X 0,Y 284.491,Z 405.045,A -85,B 0,C 180,E1 -17268.601,E2 -17268.601} C_VEL
LIN {X 0,Y 284.626,Z 405.031,A -85,B 0,C 180,E1 -17271.48,E2 -17271.48} C_VEL
LIN {X 0,Y 284.597,Z 405.034,A -85,B 0,C 180,E1 -17274.331,E2 -17274.331} C_VEL
LIN {X 0,Y 284.859,Z 405.001,A -85,B 0,C 180,E1 -17278.586,E2 -17278.586} C_VEL
LIN {X 0,Y 284.859,Z 405.004,A -85,B 0,C 180,E1 -17281.414,E2 -17281.414} C_VEL
LIN {X 0,Y 284.736,Z 405.017,A -85,B 0,C 180,E1 -17282.877,E2 -17282.877} C_VEL
LIN {X 0,Y 283.888,Z 405.124,A -85,B 0,C 180,E1 -17284.056,E2 -17284.056} C_VEL
LIN {X 0,Y 280.975,Z 405.486,A -85,B 0,C 180,E1 -17285.978,E2 -17285.978} C_VEL
LIN {X 0,Y 278.643,Z 405.779,A -85,B 0,C 180,E1 -17287.54,E2 -17287.54} C_VEL
LIN {X 0,Y 277.692,Z 405.894,A -85,B 0,C 180,E1 -17288.749,E2 -17288.749} C_VEL
LIN {X 0,Y 277.635,Z 405.903,A -85,B 0,C 180,E1 -17289.158,E2 -17289.158} C_VEL
LIN {X 0,Y 277.423,Z 405.929,A -85,B 0,C 180,E1 -17293.179,E2 -17293.179} C_VEL
LIN {X 0,Y 277.409,Z 405.927,A -85,B 0,C 180,E1 -17296.181,E2 -17296.181} C_VEL
LIN {X 0,Y 277.348,Z 405.935,A -85,B 0,C 180,E1 -17300.35,E2 -17300.35} C_VEL
LIN {X 0,Y 277.323,Z 405.94,A -85,B 0,C 180,E1 -17304.17,E2 -17304.17} C_VEL
LIN {X 0,Y 277.327,Z 405.942,A -85,B 0,C 180,E1 -17307.504,E2 -17307.504} C_VEL
LIN {X 0,Y 277.275,Z 405.947,A -85,B 0,C 180,E1 -17310.481,E2 -17310.481} C_VEL
LIN {X 0,Y 277.25,Z 405.951,A -85,B 0,C 180,E1 -17313.895,E2 -17313.895} C_VEL
LIN {X 0,Y 277.292,Z 406.005,A -85,B 0,C 180,E1 -17317.239,E2 -17317.239} C_VEL
LIN {X 0,Y 277.996,Z 410.027,A -85,B 0,C 180,E1 -17321.095,E2 -17321.095} C_VEL
LIN {X 0,Y 278.864,Z 414.566,A -85,B 0,C 180,E1 -17325.116,E2 -17325.116} C_VEL
LIN {X 0,Y 279.753,Z 419.584,A -85,B 0,C 180,E1 -17329.218,E2 -17329.218} C_VEL
LIN {X 0,Y 280.245,Z 423.346,A -85,B 0,C 180,E1 -17332.09,E2 -17332.09} C_VEL
LIN {X 0,Y 280.26,Z 425.091,A -85,B 0,C 180,E1 -17333.365,E2 -17333.365} C_VEL
LIN {X 0,Y 279.467,Z 429.459,A -85,B 0,C 180,E1 -17336.409,E2 -17336.409} C_VEL
LIN {X 0,Y 278.362,Z 435.466,A -85,B 0,C 180,E1 -17340.506,E2 -17340.506} C_VEL
LIN {X 0,Y 277.614,Z 439.838,A -85,B 0,C 180,E1 -17343.454,E2 -17343.454} C_VEL
LIN {X 0,Y 280.651,Z 453.726,A -85,B 0,C 180,E1 -17344.42,E2 -17344.42} C_VEL
LIN {X 0,Y 282.617,Z 465.749,A -85,B 0,C 180,E1 -17345.469,E2 -17345.469} C_VEL
LIN {X 0,Y 283.782,Z 478.485,A -85,B 0,C 180,E1 -17346.801,E2 -17346.801} C_VEL
LIN {X 0,Y 284.184,Z 489.745,A -85,B 0,C 180,E1 -17348.225,E2 -17348.225} C_VEL
LIN {X 0,Y 284.026,Z 493.687,A -85,B 0,C 180,E1 -17348.784,E2 -17348.784} C_VEL
LIN {X 0,Y 282.137,Z 503.894,A -85,B 0,C 180,E1 -17350.349,E2 -17350.349} C_VEL
LIN {X 0,Y 280.303,Z 514.007,A -85,B 0,C 180,E1 -17352.32,E2 -17352.32} C_VEL
LIN {X 0,Y 279.155,Z 520.726,A -85,B 0,C 180,E1 -17353.922,E2 -17353.922} C_VEL
LIN {X 0,Y 277.704,Z 528.205,A -85,B 0,C 180,E1 -17356.088,E2 -17356.088} C_VEL
LIN {X 0,Y 276.629,Z 534.224,A -85,B 0,C 180,E1 -17358.273,E2 -17358.273} C_VEL
LIN {X 0,Y 275.985,Z 538.995,A -85,B 0,C 180,E1 -17360.472,E2 -17360.472} C_VEL
LIN {X 0,Y 275.61,Z 542.648,A -85,B 0,C 180,E1 -17362.675,E2 -17362.675} C_VEL
LIN {X 0,Y 275.486,Z 544.634,A -85,B 0,C 180,E1 -17364.235,E2 -17364.235} C_VEL
LIN {X 0,Y 275.417,Z 546.969,A -85,B 0,C 180,E1 -17367.074,E2 -17367.074} C_VEL
LIN {X 0,Y 275.417,Z 547.587,A -85,B 0,C 180,E1 -17368.538,E2 -17368.538} C_VEL
LIN {X 0,Y 275.515,Z 547.811,A -85,B 0,C 180,E1 -17370,E2 -17370} C_VEL
LIN {X 0,Y 275.435,Z 547.583,A -85,B 0,C 180,E1 -17371.462,E2 -17371.462} C_VEL
LIN {X 0,Y 275.417,Z 546.961,A -85,B 0,C 180,E1 -17372.925,E2 -17372.925} C_VEL
LIN {X 0,Y 275.49,Z 544.612,A -85,B 0,C 180,E1 -17375.773,E2 -17375.773} C_VEL
LIN {X 0,Y 275.698,Z 541.536,A -85,B 0,C 180,E1 -17378.06,E2 -17378.06} C_VEL
LIN {X 0,Y 276.181,Z 537.509,A -85,B 0,C 180,E1 -17380.261,E2 -17380.261} C_VEL
LIN {X 0,Y 277.09,Z 531.33,A -85,B 0,C 180,E1 -17382.822,E2 -17382.822} C_VEL
LIN {X 0,Y 278.42,Z 524.606,A -85,B 0,C 180,E1 -17384.995,E2 -17384.995} C_VEL
LIN {X 0,Y 280.003,Z 516.268,A -85,B 0,C 180,E1 -17387.153,E2 -17387.153} C_VEL
LIN {X 0,Y 281.419,Z 507.718,A -85,B 0,C 180,E1 -17388.945,E2 -17388.945} C_VEL
LIN {X 0,Y 283.35,Z 497.183,A -85,B 0,C 180,E1 -17390.698,E2 -17390.698} C_VEL
LIN {X 0,Y 284.216,Z 490.94,A -85,B 0,C 180,E1 -17391.581,E2 -17391.581} C_VEL
LIN {X 0,Y 283.846,Z 479.583,A -85,B 0,C 180,E1 -17393.054,E2 -17393.054} C_VEL
LIN {X 0,Y 282.817,Z 468.091,A -85,B 0,C 180,E1 -17394.29,E2 -17394.29} C_VEL
LIN {X 0,Y 281.053,Z 455.747,A -85,B 0,C 180,E1 -17395.388,E2 -17395.388} C_VEL
LIN {X 0,Y 278.084,Z 442.298,A -85,B 0,C 180,E1 -17396.38,E2 -17396.38} C_VEL
LIN {X 0,Y 277.608,Z 439.802,A -85,B 0,C 180,E1 -17396.525,E2 -17396.525} C_VEL
LIN {X 0,Y 278.727,Z 433.245,A -85,B 0,C 180,E1 -17400.985,E2 -17400.985} C_VEL
LIN {X 0,Y 279.966,Z 426.998,A -85,B 0,C 180,E1 -17405.266,E2 -17405.266} C_VEL
LIN {X 0,Y 280.316,Z 424.544,A -85,B 0,C 180,E1 -17406.993,E2 -17406.993} C_VEL
LIN {X 0,Y 279.975,Z 420.804,A -85,B 0,C 180,E1 -17409.799,E2 -17409.799} C_VEL
LIN {X 0,Y 279.249,Z 416.578,A -85,B 0,C 180,E1 -17413.125,E2 -17413.125} C_VEL
LIN {X 0,Y 278.336,Z 411.968,A -85,B 0,C 180,E1 -17417.076,E2 -17417.076} C_VEL
LIN {X 0,Y 277.638,Z 408.031,A -85,B 0,C 180,E1 -17420.74,E2 -17420.74} C_VEL
LIN {X 0,Y 277.272,Z 405.947,A -85,B 0,C 180,E1 -17422.983,E2 -17422.983} C_VEL
LIN {X 0,Y 277.255,Z 405.949,A -85,B 0,C 180,E1 -17426.773,E2 -17426.773} C_VEL
LIN {X 0,Y 277.288,Z 405.946,A -85,B 0,C 180,E1 -17431.212,E2 -17431.212} C_VEL
LIN {X 0,Y 277.314,Z 405.942,A -85,B 0,C 180,E1 -17434.48,E2 -17434.48} C_VEL
LIN {X 0,Y 277.288,Z 405.943,A -85,B 0,C 180,E1 -17437.655,E2 -17437.655} C_VEL
LIN {X 0,Y 277.347,Z 405.938,A -85,B 0,C 180,E1 -17440.766,E2 -17440.766} C_VEL
LIN {X 0,Y 277.438,Z 405.926,A -85,B 0,C 180,E1 -17445.326,E2 -17445.326} C_VEL
LIN {X 0,Y 277.51,Z 405.916,A -85,B 0,C 180,E1 -17449.789,E2 -17449.789} C_VEL
LIN {X 0,Y 277.656,Z 405.9,A -85,B 0,C 180,E1 -17452.729,E2 -17452.729} C_VEL
LIN {X 0,Y 277.824,Z 405.878,A -85,B 0,C 180,E1 -17458.551,E2 -17458.551} C_VEL
LIN {X 0,Y 277.824,Z 405.875,A -85,B 0,C 180,E1 -17461.45,E2 -17461.45} C_VEL
LIN {X 0,Y 277.656,Z 405.896,A -85,B 0,C 180,E1 -17467.271,E2 -17467.271} C_VEL
LIN {X 0,Y 277.509,Z 405.918,A -85,B 0,C 180,E1 -17470.211,E2 -17470.211} C_VEL
LIN {X 0,Y 277.437,Z 405.925,A -85,B 0,C 180,E1 -17474.674,E2 -17474.674} C_VEL
LIN {X 0,Y 277.347,Z 405.935,A -85,B 0,C 180,E1 -17479.234,E2 -17479.234} C_VEL
LIN {X 0,Y 277.294,Z 405.944,A -85,B 0,C 180,E1 -17484.158,E2 -17484.158} C_VEL
LIN {X 0,Y 277.326,Z 405.939,A -85,B 0,C 180,E1 -17487.504,E2 -17487.504} C_VEL
LIN {X 0,Y 277.274,Z 405.946,A -85,B 0,C 180,E1 -17490.481,E2 -17490.481} C_VEL
LIN {X 0,Y 277.256,Z 405.949,A -85,B 0,C 180,E1 -17493.895,E2 -17493.895} C_VEL
LIN {X 0,Y 277.283,Z 405.943,A -85,B 0,C 180,E1 -17497.467,E2 -17497.467} C_VEL
LIN {X 0,Y 277.217,Z 405.952,A -85,B 0,C 180,E1 -17501.235,E2 -17501.235} C_VEL
LIN {X 0,Y 277.249,Z 405.95,A -85,B 0,C 180,E1 -17505.217,E2 -17505.217} C_VEL
LIN {X 0,Y 277.297,Z 405.945,A -85,B 0,C 180,E1 -17509.495,E2 -17509.495} C_VEL
LIN {X 0,Y 277.226,Z 405.954,A -85,B 0,C 180,E1 -17512.524,E2 -17512.524} C_VEL
LIN {X 0,Y 276.932,Z 405.994,A -85,B 0,C 180,E1 -17516.06,E2 -17516.06} C_VEL
LIN {X 0,Y 276.887,Z 406.951,A -85,B 0,C 180,E1 -17517.79,E2 -17517.79} C_VEL
LIN {X 0,Y 276.755,Z 409.454,A -85,B 0,C 180,E1 -17521.152,E2 -17521.152} C_VEL
LIN {X 0,Y 276.7,Z 411.295,A -85,B 0,C 180,E1 -17523.489,E2 -17523.489} C_VEL
LIN {X 0,Y 281.391,Z 424.644,A -85,B 0,C 180,E1 -17524.683,E2 -17524.683} C_VEL
LIN {X 0,Y 284.793,Z 436.522,A -85,B 0,C 180,E1 -17525.934,E2 -17525.934} C_VEL
LIN {X 0,Y 287.159,Z 448.006,A -85,B 0,C 180,E1 -17527.327,E2 -17527.327} C_VEL
LIN {X 0,Y 287.207,Z 451.126,A -85,B 0,C 180,E1 -17527.71,E2 -17527.71} C_VEL
LIN {X 0,Y 285.622,Z 462.139,A -85,B 0,C 180,E1 -17529.098,E2 -17529.098} C_VEL
LIN {X 0,Y 284.231,Z 471.035,A -85,B 0,C 180,E1 -17530.5,E2 -17530.5} C_VEL
LIN {X 0,Y 282.544,Z 480.167,A -85,B 0,C 180,E1 -17532.26,E2 -17532.26} C_VEL
LIN {X 0,Y 280.732,Z 489.036,A -85,B 0,C 180,E1 -17534.388,E2 -17534.388} C_VEL
LIN {X 0,Y 279.339,Z 496.161,A -85,B 0,C 180,E1 -17536.543,E2 -17536.543} C_VEL
LIN {X 0,Y 278.195,Z 500.974,A -85,B 0,C 180,E1 -17538.34,E2 -17538.34} C_VEL
LIN {X 0,Y 277.287,Z 505.635,A -85,B 0,C 180,E1 -17540.518,E2 -17540.518} C_VEL
LIN {X 0,Y 276.591,Z 509.2,A -85,B 0,C 180,E1 -17542.701,E2 -17542.701} C_VEL
LIN {X 0,Y 276.22,Z 511.043,A -85,B 0,C 180,E1 -17544.159,E2 -17544.159} C_VEL
LIN {X 0,Y 275.819,Z 513.408,A -85,B 0,C 180,E1 -17547.079,E2 -17547.079} C_VEL
LIN {X 0,Y 275.665,Z 514.242,A -85,B 0,C 180,E1 -17550,E2 -17550} C_VEL
LIN {X 0,Y 275.689,Z 514.051,A -85,B 0,C 180,E1 -17551.461,E2 -17551.461} C_VEL
LIN {X 0,Y 275.8,Z 513.469,A -85,B 0,C 180,E1 -17552.921,E2 -17552.921} C_VEL
LIN {X 0,Y 276.22,Z 511.163,A -85,B 0,C 180,E1 -17555.842,E2 -17555.842} C_VEL
LIN {X 0,Y 276.708,Z 508.527,A -85,B 0,C 180,E1 -17557.883,E2 -17557.883} C_VEL
LIN {X 0,Y 277.495,Z 504.455,A -85,B 0,C 180,E1 -17560.212,E2 -17560.212} C_VEL
LIN {X 0,Y 278.584,Z 499.464,A -85,B 0,C 180,E1 -17562.383,E2 -17562.383} C_VEL
LIN {X 0,Y 279.897,Z 493.177,A -85,B 0,C 180,E1 -17564.542,E2 -17564.542} C_VEL
LIN {X 0,Y 281.504,Z 485.303,A -85,B 0,C 180,E1 -17566.685,E2 -17566.685} C_VEL
LIN {X 0,Y 283.569,Z 475.49,A -85,B 0,C 180,E1 -17568.796,E2 -17568.796} C_VEL
LIN {X 0,Y 285.053,Z 465.857,A -85,B 0,C 180,E1 -17570.463,E2 -17570.463} C_VEL
LIN {X 0,Y 286.696,Z 454.994,A -85,B 0,C 180,E1 -17571.953,E2 -17571.953} C_VEL
LIN {X 0,Y 287.309,Z 448.963,A -85,B 0,C 180,E1 -17572.661,E2 -17572.661} C_VEL
LIN {X 0,Y 285.211,Z 438.377,A -85,B 0,C 180,E1 -17573.978,E2 -17573.978} C_VEL
LIN {X 0,Y 282.421,Z 427.984,A -85,B 0,C 180,E1 -17575.11,E2 -17575.11} C_VEL
LIN {X 0,Y 278.546,Z 416.579,A -85,B 0,C 180,E1 -17576.198,E2 -17576.198} C_VEL
LIN {X 0,Y 276.702,Z 411.233,A -85,B 0,C 180,E1 -17576.632,E2 -17576.632} C_VEL
LIN {X 0,Y 276.871,Z 408.271,A -85,B 0,C 180,E1 -17580.509,E2 -17580.509} C_VEL
LIN {X 0,Y 276.949,Z 405.989,A -85,B 0,C 180,E1 -17583.938,E2 -17583.938} C_VEL
LIN {X 0,Y 277.203,Z 405.955,A -85,B 0,C 180,E1 -17587.48,E2 -17587.48} C_VEL
LIN {X 0,Y 277.212,Z 405.953,A -85,B 0,C 180,E1 -17591.237,E2 -17591.237} C_VEL
LIN {X 0,Y 277.203,Z 405.952,A -85,B 0,C 180,E1 -17595.227,E2 -17595.227} C_VEL
LIN {X 0,Y 277.225,Z 405.951,A -85,B 0,C 180,E1 -17599.512,E2 -17599.512} C_VEL
LIN {X 0,Y 277.285,Z 405.946,A -85,B 0,C 180,E1 -17602.533,E2 -17602.533} C_VEL
LIN {X 0,Y 277.257,Z 405.949,A -85,B 0,C 180,E1 -17606.105,E2 -17606.105} C_VEL
LIN {X 0,Y 277.264,Z 405.947,A -85,B 0,C 180,E1 -17609.539,E2 -17609.539} C_VEL
LIN {X 0,Y 277.36,Z 405.934,A -85,B 0,C 180,E1 -17612.864,E2 -17612.864} C_VEL
LIN {X 0,Y 277.301,Z 405.945,A -85,B 0,C 180,E1 -17616.077,E2 -17616.077} C_VEL
LIN {X 0,Y 277.348,Z 405.935,A -85,B 0,C 180,E1 -17620.766,E2 -17620.766} C_VEL
LIN {X 0,Y 277.439,Z 405.925,A -85,B 0,C 180,E1 -17625.326,E2 -17625.326} C_VEL
LIN {X 0,Y 277.464,Z 405.924,A -85,B 0,C 180,E1 -17629.787,E2 -17629.787} C_VEL
LIN {X 0,Y 277.633,Z 405.9,A -85,B 0,C 180,E1 -17632.728,E2 -17632.728} C_VEL
LIN {X 0,Y 277.824,Z 405.877,A -85,B 0,C 180,E1 -17638.55,E2 -17638.55} C_VEL
LIN {X 0,Y 277.825,Z 405.88,A -85,B 0,C 180,E1 -17641.449,E2 -17641.449} C_VEL
LIN {X 0,Y 277.658,Z 405.899,A -85,B 0,C 180,E1 -17647.271,E2 -17647.271} C_VEL
LIN {X 0,Y 277.635,Z 405.903,A -85,B 0,C 180,E1 -17649.158,E2 -17649.158} C_VEL
LIN {X 0,Y 276.999,Z 405.987,A -85,B 0,C 180,E1 -17650.367,E2 -17650.367} C_VEL
LIN {X 0,Y 274.081,Z 406.351,A -85,B 0,C 180,E1 -17652.333,E2 -17652.333} C_VEL
LIN {X 0,Y 271.567,Z 406.659,A -85,B 0,C 180,E1 -17653.931,E2 -17653.931} C_VEL
LIN {X 0,Y 270.478,Z 406.794,A -85,B 0,C 180,E1 -17655.172,E2 -17655.172} C_VEL
LIN {X 0,Y 270.386,Z 406.802,A -85,B 0,C 180,E1 -17655.594,E2 -17655.594} C_VEL
LIN {X 0,Y 270.305,Z 406.814,A -85,B 0,C 180,E1 -17659.755,E2 -17659.755} C_VEL
LIN {X 0,Y 270.277,Z 406.818,A -85,B 0,C 180,E1 -17664.585,E2 -17664.585} C_VEL
LIN {X 0,Y 270.273,Z 406.818,A -85,B 0,C 180,E1 -17667.909,E2 -17667.909} C_VEL
LIN {X 0,Y 270.187,Z 406.832,A -85,B 0,C 180,E1 -17671.348,E2 -17671.348} C_VEL
LIN {X 0,Y 270.205,Z 406.825,A -85,B 0,C 180,E1 -17674.905,E2 -17674.905} C_VEL
LIN {X 0,Y 270.26,Z 406.937,A -85,B 0,C 180,E1 -17676.586,E2 -17676.586} C_VEL
LIN {X 0,Y 270.91,Z 410.795,A -85,B 0,C 180,E1 -17680.433,E2 -17680.433} C_VEL
LIN {X 0,Y 271.72,Z 414.963,A -85,B 0,C 180,E1 -17684.295,E2 -17684.295} C_VEL
LIN {X 0,Y 272.565,Z 419.793,A -85,B 0,C 180,E1 -17688.396,E2 -17688.396} C_VEL
LIN {X 0,Y 273.05,Z 422.46,A -85,B 0,C 180,E1 -17690.549,E2 -17690.549} C_VEL
LIN {X 0,Y 273.26,Z 425.485,A -85,B 0,C 180,E1 -17692.872,E2 -17692.872} C_VEL
LIN {X 0,Y 272.662,Z 429.208,A -85,B 0,C 180,E1 -17695.57,E2 -17695.57} C_VEL
LIN {X 0,Y 271.472,Z 435.034,A -85,B 0,C 180,E1 -17699.68,E2 -17699.68} C_VEL
LIN {X 0,Y 270.688,Z 439.39,A -85,B 0,C 180,E1 -17702.719,E2 -17702.719} C_VEL
LIN {X 0,Y 273.761,Z 453.1,A -85,B 0,C 180,E1 -17703.717,E2 -17703.717} C_VEL
LIN {X 0,Y 275.903,Z 466.143,A -85,B 0,C 180,E1 -17704.905,E2 -17704.905} C_VEL
LIN {X 0,Y 276.995,Z 477.988,A -85,B 0,C 180,E1 -17706.192,E2 -17706.192} C_VEL
LIN {X 0,Y 277.399,Z 489.303,A -85,B 0,C 180,E1 -17707.664,E2 -17707.664} C_VEL
LIN {X 0,Y 277.191,Z 494.52,A -85,B 0,C 180,E1 -17708.43,E2 -17708.43} C_VEL
LIN {X 0,Y 275.061,Z 505.429,A -85,B 0,C 180,E1 -17710.211,E2 -17710.211} C_VEL
LIN {X 0,Y 273.371,Z 514.312,A -85,B 0,C 180,E1 -17712.031,E2 -17712.031} C_VEL
LIN {X 0,Y 272.004,Z 521.659,A -85,B 0,C 180,E1 -17713.873,E2 -17713.873} C_VEL
LIN {X 0,Y 270.583,Z 528.898,A -85,B 0,C 180,E1 -17716.098,E2 -17716.098} C_VEL
LIN {X 0,Y 269.628,Z 533.789,A -85,B 0,C 180,E1 -17717.964,E2 -17717.964} C_VEL
LIN {X 0,Y 268.961,Z 538.562,A -85,B 0,C 180,E1 -17720.221,E2 -17720.221} C_VEL
LIN {X 0,Y 268.54,Z 542.215,A -85,B 0,C 180,E1 -17722.481,E2 -17722.481} C_VEL
LIN {X 0,Y 268.415,Z 544.369,A -85,B 0,C 180,E1 -17724.251,E2 -17724.251} C_VEL
LIN {X 0,Y 268.346,Z 546.538,A -85,B 0,C 180,E1 -17726.997,E2 -17726.997} C_VEL
LIN {X 0,Y 268.337,Z 547.156,A -85,B 0,C 180,E1 -17728.499,E2 -17728.499} C_VEL
LIN {X 0,Y 268.428,Z 547.379,A -85,B 0,C 180,E1 -17730,E2 -17730} C_VEL
LIN {X 0,Y 268.353,Z 547.152,A -85,B 0,C 180,E1 -17731.501,E2 -17731.501} C_VEL
LIN {X 0,Y 268.346,Z 546.529,A -85,B 0,C 180,E1 -17733.002,E2 -17733.002} C_VEL
LIN {X 0,Y 268.415,Z 544.353,A -85,B 0,C 180,E1 -17735.75,E2 -17735.75} C_VEL
LIN {X 0,Y 268.627,Z 541.1,A -85,B 0,C 180,E1 -17738.273,E2 -17738.273} C_VEL
LIN {X 0,Y 269.158,Z 537.073,A -85,B 0,C 180,E1 -17740.532,E2 -17740.532} C_VEL
LIN {X 0,Y 270.135,Z 530.894,A -85,B 0,C 180,E1 -17743.158,E2 -17743.158} C_VEL
LIN {X 0,Y 271.493,Z 524.167,A -85,B 0,C 180,E1 -17745.387,E2 -17745.387} C_VEL
LIN {X 0,Y 273.045,Z 516.492,A -85,B 0,C 180,E1 -17747.434,E2 -17747.434} C_VEL
LIN {X 0,Y 274.669,Z 507.28,A -85,B 0,C 180,E1 -17749.429,E2 -17749.429} C_VEL
LIN {X 0,Y 276.719,Z 496.747,A -85,B 0,C 180,E1 -17751.218,E2 -17751.218} C_VEL
LIN {X 0,Y 277.396,Z 491.801,A -85,B 0,C 180,E1 -17751.944,E2 -17751.944} C_VEL
LIN {X 0,Y 277.094,Z 480.342,A -85,B 0,C 180,E1 -17753.504,E2 -17753.504} C_VEL
LIN {X 0,Y 276.126,Z 468.361,A -85,B 0,C 180,E1 -17754.855,E2 -17754.855} C_VEL
LIN {X 0,Y 274.399,Z 456.569,A -85,B 0,C 180,E1 -17755.964,E2 -17755.964} C_VEL
LIN {X 0,Y 271.548,Z 443.294,A -85,B 0,C 180,E1 -17757,E2 -17757} C_VEL
LIN {X 0,Y 270.678,Z 439.31,A -85,B 0,C 180,E1 -17757.272,E2 -17757.272} C_VEL
LIN {X 0,Y 271.692,Z 433.799,A -85,B 0,C 180,E1 -17761.155,E2 -17761.155} C_VEL
LIN {X 0,Y 272.949,Z 427.803,A -85,B 0,C 180,E1 -17765.404,E2 -17765.404} C_VEL
LIN {X 0,Y 273.283,Z 425.42,A -85,B 0,C 180,E1 -17767.134,E2 -17767.134} C_VEL
LIN {X 0,Y 272.924,Z 421.635,A -85,B 0,C 180,E1 -17770.073,E2 -17770.073} C_VEL
LIN {X 0,Y 271.994,Z 416.602,A -85,B 0,C 180,E1 -17774.239,E2 -17774.239} C_VEL
LIN {X 0,Y 271.081,Z 411.607,A -85,B 0,C 180,E1 -17778.751,E2 -17778.751} C_VEL
LIN {X 0,Y 270.589,Z 408.789,A -85,B 0,C 180,E1 -17781.439,E2 -17781.439} C_VEL
LIN {X 0,Y 270.244,Z 406.824,A -85,B 0,C 180,E1 -17783.56,E2 -17783.56} C_VEL
LIN {X 0,Y 270.204,Z 406.828,A -85,B 0,C 180,E1 -17786.893,E2 -17786.893} C_VEL
LIN {X 0,Y 270.229,Z 406.825,A -85,B 0,C 180,E1 -17790.387,E2 -17790.387} C_VEL
LIN {X 0,Y 270.264,Z 406.819,A -85,B 0,C 180,E1 -17793.764,E2 -17793.764} C_VEL
LIN {X 0,Y 270.236,Z 406.823,A -85,B 0,C 180,E1 -17797.039,E2 -17797.039} C_VEL
LIN {X 0,Y 270.304,Z 406.815,A -85,B 0,C 180,E1 -17800.245,E2 -17800.245} C_VEL
LIN {X 0,Y 270.406,Z 406.803,A -85,B 0,C 180,E1 -17804.936,E2 -17804.936} C_VEL
LIN {X 0,Y 270.445,Z 406.796,A -85,B 0,C 180,E1 -17809.519,E2 -17809.519} C_VEL
LIN {X 0,Y 270.614,Z 406.779,A -85,B 0,C 180,E1 -17812.539,E2 -17812.539} C_VEL
LIN {X 0,Y 270.79,Z 406.755,A -85,B 0,C 180,E1 -17818.513,E2 -17818.513} C_VEL
LIN {X 0,Y 270.79,Z 406.752,A -85,B 0,C 180,E1 -17821.487,E2 -17821.487} C_VEL
LIN {X 0,Y 270.614,Z 406.773,A -85,B 0,C 180,E1 -17827.461,E2 -17827.461} C_VEL
LIN {X 0,Y 270.444,Z 406.798,A -85,B 0,C 180,E1 -17830.481,E2 -17830.481} C_VEL
LIN {X 0,Y 270.405,Z 406.8,A -85,B 0,C 180,E1 -17835.065,E2 -17835.065} C_VEL
LIN {X 0,Y 270.303,Z 406.814,A -85,B 0,C 180,E1 -17839.756,E2 -17839.756} C_VEL
LIN {X 0,Y 270.24,Z 406.821,A -85,B 0,C 180,E1 -17844.589,E2 -17844.589} C_VEL
LIN {X 0,Y 270.272,Z 406.82,A -85,B 0,C 180,E1 -17847.909,E2 -17847.909} C_VEL
LIN {X 0,Y 270.186,Z 406.829,A -85,B 0,C 180,E1 -17851.348,E2 -17851.348} C_VEL
LIN {X 0,Y 270.226,Z 406.823,A -85,B 0,C 180,E1 -17854.902,E2 -17854.902} C_VEL
LIN {X 0,Y 270.224,Z 406.823,A -85,B 0,C 180,E1 -17858.717,E2 -17858.717} C_VEL
LIN {X 0,Y 270.191,Z 406.827,A -85,B 0,C 180,E1 -17863.255,E2 -17863.255} C_VEL
LIN {X 0,Y 270.224,Z 406.826,A -85,B 0,C 180,E1 -17867.452,E2 -17867.452} C_VEL
LIN {X 0,Y 270.209,Z 406.829,A -85,B 0,C 180,E1 -17871.374,E2 -17871.374} C_VEL
LIN {X 0,Y 269.969,Z 406.862,A -85,B 0,C 180,E1 -17875.06,E2 -17875.06} C_VEL
LIN {X 0,Y 269.884,Z 407.381,A -85,B 0,C 180,E1 -17876.848,E2 -17876.848} C_VEL
LIN {X 0,Y 269.776,Z 409.893,A -85,B 0,C 180,E1 -17880.332,E2 -17880.332} C_VEL
LIN {X 0,Y 269.703,Z 411.822,A -85,B 0,C 180,E1 -17882.752,E2 -17882.752} C_VEL
LIN {X 0,Y 274.358,Z 424.787,A -85,B 0,C 180,E1 -17883.963,E2 -17883.963} C_VEL
LIN {X 0,Y 277.718,Z 436.235,A -85,B 0,C 180,E1 -17885.212,E2 -17885.212} C_VEL
LIN {X 0,Y 280.005,Z 446.77,A -85,B 0,C 180,E1 -17886.518,E2 -17886.518} C_VEL
LIN {X 0,Y 280.659,Z 451.564,A -85,B 0,C 180,E1 -17887.161,E2 -17887.161} C_VEL
LIN {X 0,Y 279.027,Z 462.574,A -85,B 0,C 180,E1 -17888.58,E2 -17888.58} C_VEL
LIN {X 0,Y 277.565,Z 471.515,A -85,B 0,C 180,E1 -17890.021,E2 -17890.021} C_VEL
LIN {X 0,Y 275.793,Z 480.603,A -85,B 0,C 180,E1 -17891.81,E2 -17891.81} C_VEL
LIN {X 0,Y 273.917,Z 489.47,A -85,B 0,C 180,E1 -17893.989,E2 -17893.989} C_VEL
LIN {X 0,Y 272.453,Z 496.595,A -85,B 0,C 180,E1 -17896.196,E2 -17896.196} C_VEL
LIN {X 0,Y 271.26,Z 501.407,A -85,B 0,C 180,E1 -17898.038,E2 -17898.038} C_VEL
LIN {X 0,Y 270.283,Z 506.068,A -85,B 0,C 180,E1 -17900.27,E2 -17900.27} C_VEL
LIN {X 0,Y 269.555,Z 509.633,A -85,B 0,C 180,E1 -17902.51,E2 -17902.51} C_VEL
LIN {X 0,Y 269.189,Z 511.474,A -85,B 0,C 180,E1 -17904.006,E2 -17904.006} C_VEL
LIN {X 0,Y 268.738,Z 513.84,A -85,B 0,C 180,E1 -17907.002,E2 -17907.002} C_VEL
LIN {X 0,Y 268.579,Z 514.674,A -85,B 0,C 180,E1 -17910,E2 -17910} C_VEL
LIN {X 0,Y 268.604,Z 514.483,A -85,B 0,C 180,E1 -17911.499,E2 -17911.499} C_VEL
LIN {X 0,Y 268.884,Z 512.941,A -85,B 0,C 180,E1 -17914.498,E2 -17914.498} C_VEL
LIN {X 0,Y 269.189,Z 511.592,A -85,B 0,C 180,E1 -17915.995,E2 -17915.995} C_VEL
LIN {X 0,Y 269.649,Z 509.169,A -85,B 0,C 180,E1 -17917.938,E2 -17917.938} C_VEL
LIN {X 0,Y 270.525,Z 504.885,A -85,B 0,C 180,E1 -17920.478,E2 -17920.478} C_VEL
LIN {X 0,Y 271.683,Z 499.893,A -85,B 0,C 180,E1 -17922.702,E2 -17922.702} C_VEL
LIN {X 0,Y 273.037,Z 493.606,A -85,B 0,C 180,E1 -17924.916,E2 -17924.916} C_VEL
LIN {X 0,Y 274.738,Z 485.731,A -85,B 0,C 180,E1 -17927.109,E2 -17927.109} C_VEL
LIN {X 0,Y 276.867,Z 475.918,A -85,B 0,C 180,E1 -17929.269,E2 -17929.269} C_VEL
LIN {X 0,Y 278.366,Z 466.706,A -85,B 0,C 180,E1 -17930.908,E2 -17930.908} C_VEL
LIN {X 0,Y 280.16,Z 455.419,A -85,B 0,C 180,E1 -17932.492,E2 -17932.492} C_VEL
LIN {X 0,Y 280.69,Z 450.953,A -85,B 0,C 180,E1 -17933.031,E2 -17933.031} C_VEL
LIN {X 0,Y 278.785,Z 440.7,A -85,B 0,C 180,E1 -17934.375,E2 -17934.375} C_VEL
LIN {X 0,Y 275.85,Z 429.502,A -85,B 0,C 180,E1 -17935.666,E2 -17935.666} C_VEL
LIN {X 0,Y 271.894,Z 417.635,A -85,B 0,C 180,E1 -17936.858,E2 -17936.858} C_VEL
LIN {X 0,Y 269.696,Z 411.679,A -85,B 0,C 180,E1 -17937.39,E2 -17937.39} C_VEL
LIN {X 0,Y 269.842,Z 408.717,A -85,B 0,C 180,E1 -17941.393,E2 -17941.393} C_VEL
LIN {X 0,Y 269.936,Z 407.178,A -85,B 0,C 180,E1 -17943.576,E2 -17943.576} C_VEL
LIN {X 0,Y 270.097,Z 406.842,A -85,B 0,C 180,E1 -17946.761,E2 -17946.761} C_VEL
LIN {X 0,Y 270.177,Z 406.832,A -85,B 0,C 180,E1 -17950.566,E2 -17950.566} C_VEL
LIN {X 0,Y 270.155,Z 406.833,A -85,B 0,C 180,E1 -17954.62,E2 -17954.62} C_VEL
LIN {X 0,Y 270.172,Z 406.83,A -85,B 0,C 180,E1 -17958.972,E2 -17958.972} C_VEL
LIN {X 0,Y 270.21,Z 406.822,A -85,B 0,C 180,E1 -17961.374,E2 -17961.374} C_VEL
LIN {X 0,Y 270.218,Z 406.822,A -85,B 0,C 180,E1 -17965.097,E2 -17965.097} C_VEL
LIN {X 0,Y 270.203,Z 406.826,A -85,B 0,C 180,E1 -17969.131,E2 -17969.131} C_VEL
LIN {X 0,Y 270.266,Z 406.82,A -85,B 0,C 180,E1 -17972.146,E2 -17972.146} C_VEL
LIN {X 0,Y 270.241,Z 406.82,A -85,B 0,C 180,E1 -17975.538,E2 -17975.538} C_VEL
LIN {X 0,Y 270.305,Z 406.814,A -85,B 0,C 180,E1 -17980.245,E2 -17980.245} C_VEL
LIN {X 0,Y 270.407,Z 406.8,A -85,B 0,C 180,E1 -17984.935,E2 -17984.935} C_VEL
LIN {X 0,Y 270.416,Z 406.801,A -85,B 0,C 180,E1 -17989.518,E2 -17989.518} C_VEL
LIN {X 0,Y 270.589,Z 406.778,A -85,B 0,C 180,E1 -17992.538,E2 -17992.538} C_VEL
LIN {X 0,Y 270.79,Z 406.754,A -85,B 0,C 180,E1 -17998.513,E2 -17998.513} C_VEL
LIN {X 0,Y 270.791,Z 406.756,A -85,B 0,C 180,E1 -18001.487,E2 -18001.487} C_VEL
LIN {X 0,Y 270.616,Z 406.778,A -85,B 0,C 180,E1 -18007.461,E2 -18007.461} C_VEL
LIN {X 0,Y 270.446,Z 406.796,A -85,B 0,C 180,E1 -18010.481,E2 -18010.481} C_VEL
LIN {X 0,Y 270.407,Z 406.802,A -85,B 0,C 180,E1 -18015.064,E2 -18015.064} C_VEL
LIN {X 0,Y 270.386,Z 406.802,A -85,B 0,C 180,E1 -18015.594,E2 -18015.594} C_VEL
LIN {X 0,Y 269.698,Z 406.889,A -85,B 0,C 180,E1 -18016.836,E2 -18016.836} C_VEL
LIN {X 0,Y 266.791,Z 407.255,A -85,B 0,C 180,E1 -18018.858,E2 -18018.858} C_VEL
LIN {X 0,Y 264.319,Z 407.563,A -85,B 0,C 180,E1 -18020.502,E2 -18020.502} C_VEL
LIN {X 0,Y 263.246,Z 407.694,A -85,B 0,C 180,E1 -18021.779,E2 -18021.779} C_VEL
LIN {X 0,Y 263.151,Z 407.704,A -85,B 0,C 180,E1 -18022.211,E2 -18022.211} C_VEL
LIN {X 0,Y 263.211,Z 407.7,A -85,B 0,C 180,E1 -18025.291,E2 -18025.291} C_VEL
LIN {X 0,Y 263.168,Z 407.704,A -85,B 0,C 180,E1 -18028.731,E2 -18028.731} C_VEL
LIN {X 0,Y 263.135,Z 407.708,A -85,B 0,C 180,E1 -18032.288,E2 -18032.288} C_VEL
LIN {X 0,Y 263.173,Z 407.724,A -85,B 0,C 180,E1 -18035.744,E2 -18035.744} C_VEL
LIN {X 0,Y 263.85,Z 411.554,A -85,B 0,C 180,E1 -18039.738,E2 -18039.738} C_VEL
LIN {X 0,Y 264.615,Z 415.666,A -85,B 0,C 180,E1 -18043.673,E2 -18043.673} C_VEL
LIN {X 0,Y 265.174,Z 418.734,A -85,B 0,C 180,E1 -18046.442,E2 -18046.442} C_VEL
LIN {X 0,Y 266.073,Z 423.74,A -85,B 0,C 180,E1 -18050.659,E2 -18050.659} C_VEL
LIN {X 0,Y 266.125,Z 427.424,A -85,B 0,C 180,E1 -18053.544,E2 -18053.544} C_VEL
LIN {X 0,Y 265.135,Z 432.224,A -85,B 0,C 180,E1 -18057.084,E2 -18057.084} C_VEL
LIN {X 0,Y 263.903,Z 438.331,A -85,B 0,C 180,E1 -18061.501,E2 -18061.501} C_VEL
LIN {X 0,Y 263.799,Z 438.941,A -85,B 0,C 180,E1 -18061.944,E2 -18061.944} C_VEL
LIN {X 0,Y 266.93,Z 452.578,A -85,B 0,C 180,E1 -18062.986,E2 -18062.986} C_VEL
LIN {X 0,Y 269.114,Z 465.693,A -85,B 0,C 180,E1 -18064.226,E2 -18064.226} C_VEL
LIN {X 0,Y 270.283,Z 478.565,A -85,B 0,C 180,E1 -18065.68,E2 -18065.68} C_VEL
LIN {X 0,Y 270.61,Z 490.189,A -85,B 0,C 180,E1 -18067.274,E2 -18067.274} C_VEL
LIN {X 0,Y 270.367,Z 495.271,A -85,B 0,C 180,E1 -18068.058,E2 -18068.058} C_VEL
LIN {X 0,Y 268.356,Z 504.997,A -85,B 0,C 180,E1 -18069.695,E2 -18069.695} C_VEL
LIN {X 0,Y 266.416,Z 514.704,A -85,B 0,C 180,E1 -18071.745,E2 -18071.745} C_VEL
LIN {X 0,Y 265.176,Z 521.228,A -85,B 0,C 180,E1 -18073.446,E2 -18073.446} C_VEL
LIN {X 0,Y 263.638,Z 528.463,A -85,B 0,C 180,E1 -18075.724,E2 -18075.724} C_VEL
LIN {X 0,Y 262.639,Z 533.355,A -85,B 0,C 180,E1 -18077.639,E2 -18077.639} C_VEL
LIN {X 0,Y 261.916,Z 538.127,A -85,B 0,C 180,E1 -18079.955,E2 -18079.955} C_VEL
LIN {X 0,Y 261.475,Z 541.781,A -85,B 0,C 180,E1 -18082.276,E2 -18082.276} C_VEL
LIN {X 0,Y 261.328,Z 544.136,A -85,B 0,C 180,E1 -18084.302,E2 -18084.302} C_VEL
LIN {X 0,Y 261.276,Z 546.107,A -85,B 0,C 180,E1 -18086.916,E2 -18086.916} C_VEL
LIN {X 0,Y 261.259,Z 546.725,A -85,B 0,C 180,E1 -18088.458,E2 -18088.458} C_VEL
LIN {X 0,Y 261.343,Z 546.948,A -85,B 0,C 180,E1 -18090,E2 -18090} C_VEL
LIN {X 0,Y 261.274,Z 546.72,A -85,B 0,C 180,E1 -18091.541,E2 -18091.541} C_VEL
LIN {X 0,Y 261.276,Z 546.098,A -85,B 0,C 180,E1 -18093.084,E2 -18093.084} C_VEL
LIN {X 0,Y 261.335,Z 544.106,A -85,B 0,C 180,E1 -18095.713,E2 -18095.713} C_VEL
LIN {X 0,Y 261.572,Z 540.665,A -85,B 0,C 180,E1 -18098.498,E2 -18098.498} C_VEL
LIN {X 0,Y 262.124,Z 536.636,A -85,B 0,C 180,E1 -18100.817,E2 -18100.817} C_VEL
LIN {X 0,Y 263.203,Z 530.458,A -85,B 0,C 180,E1 -18103.511,E2 -18103.511} C_VEL
LIN {X 0,Y 264.58,Z 523.728,A -85,B 0,C 180,E1 -18105.799,E2 -18105.799} C_VEL
LIN {X 0,Y 266.265,Z 515.747,A -85,B 0,C 180,E1 -18107.973,E2 -18107.973} C_VEL
LIN {X 0,Y 267.949,Z 506.842,A -85,B 0,C 180,E1 -18109.936,E2 -18109.936} C_VEL
LIN {X 0,Y 270.102,Z 496.31,A -85,B 0,C 180,E1 -18111.764,E2 -18111.764} C_VEL
LIN {X 0,Y 270.595,Z 492.662,A -85,B 0,C 180,E1 -18112.324,E2 -18112.324} C_VEL
LIN {X 0,Y 270.401,Z 482.217,A -85,B 0,C 180,E1 -18113.827,E2 -18113.827} C_VEL
LIN {X 0,Y 269.622,Z 471.127,A -85,B 0,C 180,E1 -18115.174,E2 -18115.174} C_VEL
LIN {X 0,Y 268.18,Z 459.403,A -85,B 0,C 180,E1 -18116.369,E2 -18116.369} C_VEL
LIN {X 0,Y 265.575,Z 446.672,A -85,B 0,C 180,E1 -18117.477,E2 -18117.477} C_VEL
LIN {X 0,Y 263.782,Z 438.868,A -85,B 0,C 180,E1 -18118.049,E2 -18118.049} C_VEL
LIN {X 0,Y 264.895,Z 433.37,A -85,B 0,C 180,E1 -18122.048,E2 -18122.048} C_VEL
LIN {X 0,Y 265.924,Z 428.581,A -85,B 0,C 180,E1 -18125.551,E2 -18125.551} C_VEL
LIN {X 0,Y 266.251,Z 425.832,A -85,B 0,C 180,E1 -18127.638,E2 -18127.638} C_VEL
LIN {X 0,Y 265.959,Z 422.909,A -85,B 0,C 180,E1 -18129.975,E2 -18129.975} C_VEL
LIN {X 0,Y 265.022,Z 417.859,A -85,B 0,C 180,E1 -18134.275,E2 -18134.275} C_VEL
LIN {X 0,Y 264.183,Z 413.48,A -85,B 0,C 180,E1 -18138.312,E2 -18138.312} C_VEL
LIN {X 0,Y 263.385,Z 408.666,A -85,B 0,C 180,E1 -18143.178,E2 -18143.178} C_VEL
LIN {X 0,Y 263.172,Z 407.702,A -85,B 0,C 180,E1 -18144.256,E2 -18144.256} C_VEL
LIN {X 0,Y 263.142,Z 407.705,A -85,B 0,C 180,E1 -18148.722,E2 -18148.722} C_VEL
LIN {X 0,Y 263.194,Z 407.702,A -85,B 0,C 180,E1 -18153.003,E2 -18153.003} C_VEL
LIN {X 0,Y 263.187,Z 407.702,A -85,B 0,C 180,E1 -18156.387,E2 -18156.387} C_VEL
LIN {X 0,Y 263.266,Z 407.69,A -85,B 0,C 180,E1 -18159.694,E2 -18159.694} C_VEL
LIN {X 0,Y 263.353,Z 407.683,A -85,B 0,C 180,E1 -18164.522,E2 -18164.522} C_VEL
LIN {X 0,Y 263.377,Z 407.677,A -85,B 0,C 180,E1 -18169.235,E2 -18169.235} C_VEL
LIN {X 0,Y 263.576,Z 407.655,A -85,B 0,C 180,E1 -18172.339,E2 -18172.339} C_VEL
LIN {X 0,Y 263.754,Z 407.631,A -85,B 0,C 180,E1 -18178.473,E2 -18178.473} C_VEL
LIN {X 0,Y 263.754,Z 407.628,A -85,B 0,C 180,E1 -18181.527,E2 -18181.527} C_VEL
LIN {X 0,Y 263.576,Z 407.65,A -85,B 0,C 180,E1 -18187.662,E2 -18187.662} C_VEL
LIN {X 0,Y 263.376,Z 407.677,A -85,B 0,C 180,E1 -18190.766,E2 -18190.766} C_VEL
LIN {X 0,Y 263.353,Z 407.679,A -85,B 0,C 180,E1 -18195.478,E2 -18195.478} C_VEL
LIN {X 0,Y 263.265,Z 407.692,A -85,B 0,C 180,E1 -18200.307,E2 -18200.307} C_VEL
LIN {X 0,Y 263.195,Z 407.699,A -85,B 0,C 180,E1 -18205.293,E2 -18205.293} C_VEL
LIN {X 0,Y 263.168,Z 407.702,A -85,B 0,C 180,E1 -18208.731,E2 -18208.731} C_VEL
LIN {X 0,Y 263.135,Z 407.703,A -85,B 0,C 180,E1 -18212.288,E2 -18212.288} C_VEL
LIN {X 0,Y 263.192,Z 407.699,A -85,B 0,C 180,E1 -18215.978,E2 -18215.978} C_VEL
LIN {X 0,Y 263.119,Z 407.709,A -85,B 0,C 180,E1 -18219.87,E2 -18219.87} C_VEL
LIN {X 0,Y 263.14,Z 407.708,A -85,B 0,C 180,E1 -18223.981,E2 -18223.981} C_VEL
LIN {X 0,Y 263.175,Z 407.703,A -85,B 0,C 180,E1 -18228.394,E2 -18228.394} C_VEL
LIN {X 0,Y 263.107,Z 407.714,A -85,B 0,C 180,E1 -18232.094,E2 -18232.094} C_VEL
LIN {X 0,Y 262.86,Z 407.919,A -85,B 0,C 180,E1 -18235.98,E2 -18235.98} C_VEL
LIN {X 0,Y 262.796,Z 410.35,A -85,B 0,C 180,E1 -18239.461,E2 -18239.461} C_VEL
LIN {X 0,Y 262.667,Z 412.167,A -85,B 0,C 180,E1 -18241.928,E2 -18241.928} C_VEL
LIN {X 0,Y 263.797,Z 415.362,A -85,B 0,C 180,E1 -18242.236,E2 -18242.236} C_VEL
LIN {X 0,Y 268.166,Z 427.373,A -85,B 0,C 180,E1 -18243.465,E2 -18243.465} C_VEL
LIN {X 0,Y 271.631,Z 439.615,A -85,B 0,C 180,E1 -18244.901,E2 -18244.901} C_VEL
LIN {X 0,Y 273.795,Z 450.524,A -85,B 0,C 180,E1 -18246.362,E2 -18246.362} C_VEL
LIN {X 0,Y 273.965,Z 453.593,A -85,B 0,C 180,E1 -18246.775,E2 -18246.775} C_VEL
LIN {X 0,Y 272.155,Z 464.563,A -85,B 0,C 180,E1 -18248.274,E2 -18248.274} C_VEL
LIN {X 0,Y 270.567,Z 473.964,A -85,B 0,C 180,E1 -18249.892,E2 -18249.892} C_VEL
LIN {X 0,Y 268.709,Z 482.651,A -85,B 0,C 180,E1 -18251.708,E2 -18251.708} C_VEL
LIN {X 0,Y 266.829,Z 491.225,A -85,B 0,C 180,E1 -18253.945,E2 -18253.945} C_VEL
LIN {X 0,Y 265.332,Z 498.05,A -85,B 0,C 180,E1 -18256.209,E2 -18256.209} C_VEL
LIN {X 0,Y 263.941,Z 503.521,A -85,B 0,C 180,E1 -18258.48,E2 -18258.48} C_VEL
LIN {X 0,Y 263.039,Z 507.8,A -85,B 0,C 180,E1 -18260.775,E2 -18260.775} C_VEL
LIN {X 0,Y 262.528,Z 510.066,A -85,B 0,C 180,E1 -18262.308,E2 -18262.308} C_VEL
LIN {X 0,Y 262.16,Z 511.905,A -85,B 0,C 180,E1 -18263.844,E2 -18263.844} C_VEL
LIN {X 0,Y 261.661,Z 514.272,A -85,B 0,C 180,E1 -18266.921,E2 -18266.921} C_VEL
LIN {X 0,Y 261.493,Z 515.105,A -85,B 0,C 180,E1 -18270,E2 -18270} C_VEL
LIN {X 0,Y 261.519,Z 514.914,A -85,B 0,C 180,E1 -18271.54,E2 -18271.54} C_VEL
LIN {X 0,Y 261.831,Z 513.372,A -85,B 0,C 180,E1 -18274.619,E2 -18274.619} C_VEL
LIN {X 0,Y 262.159,Z 512.022,A -85,B 0,C 180,E1 -18276.156,E2 -18276.156} C_VEL
LIN {X 0,Y 262.59,Z 509.812,A -85,B 0,C 180,E1 -18277.996,E2 -18277.996} C_VEL
LIN {X 0,Y 263.545,Z 505.317,A -85,B 0,C 180,E1 -18280.759,E2 -18280.759} C_VEL
LIN {X 0,Y 264.777,Z 500.323,A -85,B 0,C 180,E1 -18283.039,E2 -18283.039} C_VEL
LIN {X 0,Y 266.198,Z 494.036,A -85,B 0,C 180,E1 -18285.309,E2 -18285.309} C_VEL
LIN {X 0,Y 267.991,Z 486.158,A -85,B 0,C 180,E1 -18287.553,E2 -18287.553} C_VEL
LIN {X 0,Y 270.182,Z 476.347,A -85,B 0,C 180,E1 -18289.765,E2 -18289.765} C_VEL
LIN {X 0,Y 271.931,Z 466.061,A -85,B 0,C 180,E1 -18291.61,E2 -18291.61} C_VEL
LIN {X 0,Y 273.859,Z 454.427,A -85,B 0,C 180,E1 -18293.239,E2 -18293.239} C_VEL
LIN {X 0,Y 273.948,Z 451.395,A -85,B 0,C 180,E1 -18293.632,E2 -18293.632} C_VEL
LIN {X 0,Y 271.753,Z 440.145,A -85,B 0,C 180,E1 -18295.155,E2 -18295.155} C_VEL
LIN {X 0,Y 268.308,Z 427.648,A -85,B 0,C 180,E1 -18296.625,E2 -18296.625} C_VEL
LIN {X 0,Y 263.739,Z 415.181,A -85,B 0,C 180,E1 -18297.906,E2 -18297.906} C_VEL
LIN {X 0,Y 262.697,Z 412.135,A -85,B 0,C 180,E1 -18298.182,E2 -18298.182} C_VEL
LIN {X 0,Y 262.863,Z 409.162,A -85,B 0,C 180,E1 -18302.326,E2 -18302.326} C_VEL
LIN {X 0,Y 262.912,Z 407.916,A -85,B 0,C 180,E1 -18304.15,E2 -18304.15} C_VEL
LIN {X 0,Y 263.062,Z 407.718,A -85,B 0,C 180,E1 -18307.914,E2 -18307.914} C_VEL
LIN {X 0,Y 263.126,Z 407.708,A -85,B 0,C 180,E1 -18311.893,E2 -18311.893} C_VEL
LIN {X 0,Y 263.127,Z 407.708,A -85,B 0,C 180,E1 -18316.151,E2 -18316.151} C_VEL
LIN {X 0,Y 263.118,Z 407.711,A -85,B 0,C 180,E1 -18320.13,E2 -18320.13} C_VEL
LIN {X 0,Y 263.191,Z 407.7,A -85,B 0,C 180,E1 -18324.022,E2 -18324.022} C_VEL
LIN {X 0,Y 263.137,Z 407.707,A -85,B 0,C 180,E1 -18327.712,E2 -18327.712} C_VEL
LIN {X 0,Y 263.199,Z 407.7,A -85,B 0,C 180,E1 -18331.785,E2 -18331.785} C_VEL
LIN {X 0,Y 263.204,Z 407.696,A -85,B 0,C 180,E1 -18335.212,E2 -18335.212} C_VEL
LIN {X 0,Y 263.266,Z 407.692,A -85,B 0,C 180,E1 -18339.693,E2 -18339.693} C_VEL
LIN {X 0,Y 263.355,Z 407.68,A -85,B 0,C 180,E1 -18344.522,E2 -18344.522} C_VEL
LIN {X 0,Y 263.358,Z 407.678,A -85,B 0,C 180,E1 -18349.234,E2 -18349.234} C_VEL
LIN {X 0,Y 263.548,Z 407.656,A -85,B 0,C 180,E1 -18352.338,E2 -18352.338} C_VEL
LIN {X 0,Y 263.755,Z 407.631,A -85,B 0,C 180,E1 -18358.473,E2 -18358.473} C_VEL
LIN {X 0,Y 263.755,Z 407.633,A -85,B 0,C 180,E1 -18361.527,E2 -18361.527} C_VEL
LIN {X 0,Y 263.577,Z 407.657,A -85,B 0,C 180,E1 -18367.661,E2 -18367.661} C_VEL
LIN {X 0,Y 263.379,Z 407.677,A -85,B 0,C 180,E1 -18370.765,E2 -18370.765} C_VEL
LIN {X 0,Y 263.352,Z 407.681,A -85,B 0,C 180,E1 -18375.586,E2 -18375.586} C_VEL
LIN {X 0,Y 263.267,Z 407.689,A -85,B 0,C 180,E1 -18380.306,E2 -18380.306} C_VEL
LIN {X 0,Y 263.151,Z 407.704,A -85,B 0,C 180,E1 -18382.211,E2 -18382.211} C_VEL
LIN {X 0,Y 262.471,Z 407.791,A -85,B 0,C 180,E1 -18383.488,E2 -18383.488} C_VEL
LIN {X 0,Y 259.642,Z 408.145,A -85,B 0,C 180,E1 -18385.571,E2 -18385.571} C_VEL
LIN {X 0,Y 257.242,Z 408.444,A -85,B 0,C 180,E1 -18387.264,E2 -18387.264} C_VEL
LIN {X 0,Y 256.201,Z 408.572,A -85,B 0,C 180,E1 -18388.577,E2 -18388.577} C_VEL
LIN {X 0,Y 256.11,Z 408.582,A -85,B 0,C 180,E1 -18389.022,E2 -18389.022} C_VEL
LIN {X 0,Y 256.079,Z 408.588,A -85,B 0,C 180,E1 -18393.291,E2 -18393.291} C_VEL
LIN {X 0,Y 256.158,Z 408.785,A -85,B 0,C 180,E1 -18395.181,E2 -18395.181} C_VEL
LIN {X 0,Y 256.77,Z 412.311,A -85,B 0,C 180,E1 -18399.015,E2 -18399.015} C_VEL
LIN {X 0,Y 257.511,Z 416.341,A -85,B 0,C 180,E1 -18403.024,E2 -18403.024} C_VEL
LIN {X 0,Y 258.14,Z 419.654,A -85,B 0,C 180,E1 -18406.113,E2 -18406.113} C_VEL
LIN {X 0,Y 259.024,Z 424.625,A -85,B 0,C 180,E1 -18410.465,E2 -18410.465} C_VEL
LIN {X 0,Y 259.103,Z 428.203,A -85,B 0,C 180,E1 -18413.363,E2 -18413.363} C_VEL
LIN {X 0,Y 258.091,Z 432.982,A -85,B 0,C 180,E1 -18417.001,E2 -18417.001} C_VEL
LIN {X 0,Y 256.927,Z 438.486,A -85,B 0,C 180,E1 -18421.12,E2 -18421.12} C_VEL
LIN {X 0,Y 259.661,Z 450.166,A -85,B 0,C 180,E1 -18422.044,E2 -18422.044} C_VEL
LIN {X 0,Y 261.99,Z 462.935,A -85,B 0,C 180,E1 -18423.257,E2 -18423.257} C_VEL
LIN {X 0,Y 263.201,Z 473.632,A -85,B 0,C 180,E1 -18424.454,E2 -18424.454} C_VEL
LIN {X 0,Y 263.752,Z 484.705,A -85,B 0,C 180,E1 -18425.906,E2 -18425.906} C_VEL
LIN {X 0,Y 263.751,Z 494.84,A -85,B 0,C 180,E1 -18427.478,E2 -18427.478} C_VEL
LIN {X 0,Y 261.687,Z 504.566,A -85,B 0,C 180,E1 -18429.154,E2 -18429.154} C_VEL
LIN {X 0,Y 259.812,Z 513.447,A -85,B 0,C 180,E1 -18431.058,E2 -18431.058} C_VEL
LIN {X 0,Y 258.366,Z 520.797,A -85,B 0,C 180,E1 -18432.997,E2 -18432.997} C_VEL
LIN {X 0,Y 256.727,Z 528.03,A -85,B 0,C 180,E1 -18435.331,E2 -18435.331} C_VEL
LIN {X 0,Y 255.656,Z 532.921,A -85,B 0,C 180,E1 -18437.295,E2 -18437.295} C_VEL
LIN {X 0,Y 254.876,Z 537.693,A -85,B 0,C 180,E1 -18439.675,E2 -18439.675} C_VEL
LIN {X 0,Y 254.401,Z 541.347,A -85,B 0,C 180,E1 -18442.06,E2 -18442.06} C_VEL
LIN {X 0,Y 254.229,Z 543.929,A -85,B 0,C 180,E1 -18444.384,E2 -18444.384} C_VEL
LIN {X 0,Y 254.207,Z 545.676,A -85,B 0,C 180,E1 -18446.83,E2 -18446.83} C_VEL
LIN {X 0,Y 254.184,Z 546.294,A -85,B 0,C 180,E1 -18448.415,E2 -18448.415} C_VEL
LIN {X 0,Y 254.26,Z 546.517,A -85,B 0,C 180,E1 -18450,E2 -18450} C_VEL
LIN {X 0,Y 254.197,Z 546.289,A -85,B 0,C 180,E1 -18451.584,E2 -18451.584} C_VEL
LIN {X 0,Y 254.206,Z 545.667,A -85,B 0,C 180,E1 -18453.17,E2 -18453.17} C_VEL
LIN {X 0,Y 254.23,Z 543.91,A -85,B 0,C 180,E1 -18455.618,E2 -18455.618} C_VEL
LIN {X 0,Y 254.538,Z 540.231,A -85,B 0,C 180,E1 -18458.735,E2 -18458.735} C_VEL
LIN {X 0,Y 255.11,Z 536.2,A -85,B 0,C 180,E1 -18461.119,E2 -18461.119} C_VEL
LIN {X 0,Y 256.287,Z 530.023,A -85,B 0,C 180,E1 -18463.883,E2 -18463.883} C_VEL
LIN {X 0,Y 257.708,Z 523.29,A -85,B 0,C 180,E1 -18466.232,E2 -18466.232} C_VEL
LIN {X 0,Y 259.318,Z 516.043,A -85,B 0,C 180,E1 -18468.272,E2 -18468.272} C_VEL
LIN {X 0,Y 261.247,Z 506.404,A -85,B 0,C 180,E1 -18470.47,E2 -18470.47} C_VEL
LIN {X 0,Y 263.488,Z 495.872,A -85,B 0,C 180,E1 -18472.339,E2 -18472.339} C_VEL
LIN {X 0,Y 263.848,Z 489.585,A -85,B 0,C 180,E1 -18473.342,E2 -18473.342} C_VEL
LIN {X 0,Y 263.515,Z 478.329,A -85,B 0,C 180,E1 -18474.935,E2 -18474.935} C_VEL
LIN {X 0,Y 262.448,Z 466.105,A -85,B 0,C 180,E1 -18476.369,E2 -18476.369} C_VEL
LIN {X 0,Y 260.123,Z 452.373,A -85,B 0,C 180,E1 -18477.733,E2 -18477.733} C_VEL
LIN {X 0,Y 256.991,Z 439.169,A -85,B 0,C 180,E1 -18478.805,E2 -18478.805} C_VEL
LIN {X 0,Y 256.905,Z 438.439,A -85,B 0,C 180,E1 -18478.845,E2 -18478.845} C_VEL
LIN {X 0,Y 258.096,Z 432.938,A -85,B 0,C 180,E1 -18482.998,E2 -18482.998} C_VEL
LIN {X 0,Y 259.118,Z 428.149,A -85,B 0,C 180,E1 -18486.634,E2 -18486.634} C_VEL
LIN {X 0,Y 259.049,Z 424.581,A -85,B 0,C 180,E1 -18489.531,E2 -18489.531} C_VEL
LIN {X 0,Y 258.126,Z 419.605,A -85,B 0,C 180,E1 -18493.884,E2 -18493.884} C_VEL
LIN {X 0,Y 257.373,Z 415.717,A -85,B 0,C 180,E1 -18497.5,E2 -18497.5} C_VEL
LIN {X 0,Y 256.739,Z 412.274,A -85,B 0,C 180,E1 -18500.979,E2 -18500.979} C_VEL
LIN {X 0,Y 256.487,Z 410.403,A -85,B 0,C 180,E1 -18502.928,E2 -18502.928} C_VEL
LIN {X 0,Y 256.116,Z 408.586,A -85,B 0,C 180,E1 -18505.179,E2 -18505.179} C_VEL
LIN {X 0,Y 256.094,Z 408.583,A -85,B 0,C 180,E1 -18508.573,E2 -18508.573} C_VEL
LIN {X 0,Y 256.143,Z 408.579,A -85,B 0,C 180,E1 -18512.196,E2 -18512.196} C_VEL
LIN {X 0,Y 256.169,Z 408.574,A -85,B 0,C 180,E1 -18515.699,E2 -18515.699} C_VEL
LIN {X 0,Y 256.169,Z 408.576,A -85,B 0,C 180,E1 -18519.105,E2 -18519.105} C_VEL
LIN {X 0,Y 256.302,Z 408.56,A -85,B 0,C 180,E1 -18524.085,E2 -18524.085} C_VEL
LIN {X 0,Y 256.313,Z 408.558,A -85,B 0,C 180,E1 -18528.934,E2 -18528.934} C_VEL
LIN {X 0,Y 256.543,Z 408.53,A -85,B 0,C 180,E1 -18532.127,E2 -18532.127} C_VEL
LIN {X 0,Y 256.717,Z 408.508,A -85,B 0,C 180,E1 -18538.431,E2 -18538.431} C_VEL
LIN {X 0,Y 256.717,Z 408.505,A -85,B 0,C 180,E1 -18541.569,E2 -18541.569} C_VEL
LIN {X 0,Y 256.543,Z 408.527,A -85,B 0,C 180,E1 -18547.873,E2 -18547.873} C_VEL
LIN {X 0,Y 256.312,Z 408.556,A -85,B 0,C 180,E1 -18551.066,E2 -18551.066} C_VEL
LIN {X 0,Y 256.303,Z 408.559,A -85,B 0,C 180,E1 -18555.915,E2 -18555.915} C_VEL
LIN {X 0,Y 256.165,Z 408.574,A -85,B 0,C 180,E1 -18560.895,E2 -18560.895} C_VEL
LIN {X 0,Y 256.173,Z 408.573,A -85,B 0,C 180,E1 -18565.13,E2 -18565.13} C_VEL
LIN {X 0,Y 256.106,Z 408.583,A -85,B 0,C 180,E1 -18569.601,E2 -18569.601} C_VEL
LIN {X 0,Y 256.087,Z 408.58,A -85,B 0,C 180,E1 -18573.29,E2 -18573.29} C_VEL
LIN {X 0,Y 256.13,Z 408.576,A -85,B 0,C 180,E1 -18577.275,E2 -18577.275} C_VEL
LIN {X 0,Y 256.063,Z 408.587,A -85,B 0,C 180,E1 -18581.202,E2 -18581.202} C_VEL
LIN {X 0,Y 256.078,Z 408.588,A -85,B 0,C 180,E1 -18585.526,E2 -18585.526} C_VEL
LIN {X 0,Y 256.106,Z 408.583,A -85,B 0,C 180,E1 -18588.806,E2 -18588.806} C_VEL
LIN {X 0,Y 256.029,Z 408.596,A -85,B 0,C 180,E1 -18592.85,E2 -18592.85} C_VEL
LIN {X 0,Y 255.837,Z 408.751,A -85,B 0,C 180,E1 -18595.5,E2 -18595.5} C_VEL
LIN {X 0,Y 255.795,Z 410.792,A -85,B 0,C 180,E1 -18598.532,E2 -18598.532} C_VEL
LIN {X 0,Y 255.689,Z 412.632,A -85,B 0,C 180,E1 -18601.104,E2 -18601.104} C_VEL
LIN {X 0,Y 256.822,Z 415.826,A -85,B 0,C 180,E1 -18601.412,E2 -18601.412} C_VEL
LIN {X 0,Y 261.119,Z 427.28,A -85,B 0,C 180,E1 -18602.648,E2 -18602.648} C_VEL
LIN {X 0,Y 264.462,Z 438.808,A -85,B 0,C 180,E1 -18604.036,E2 -18604.036} C_VEL
LIN {X 0,Y 266.661,Z 448.864,A -85,B 0,C 180,E1 -18605.409,E2 -18605.409} C_VEL
LIN {X 0,Y 267.418,Z 454.273,A -85,B 0,C 180,E1 -18606.206,E2 -18606.206} C_VEL
LIN {X 0,Y 265.648,Z 464.74,A -85,B 0,C 180,E1 -18607.668,E2 -18607.668} C_VEL
LIN {X 0,Y 263.921,Z 474.482,A -85,B 0,C 180,E1 -18609.381,E2 -18609.381} C_VEL
LIN {X 0,Y 261.995,Z 483.085,A -85,B 0,C 180,E1 -18611.222,E2 -18611.222} C_VEL
LIN {X 0,Y 260.037,Z 491.658,A -85,B 0,C 180,E1 -18613.514,E2 -18613.514} C_VEL
LIN {X 0,Y 258.469,Z 498.483,A -85,B 0,C 180,E1 -18615.835,E2 -18615.835} C_VEL
LIN {X 0,Y 256.997,Z 503.954,A -85,B 0,C 180,E1 -18618.165,E2 -18618.165} C_VEL
LIN {X 0,Y 256.05,Z 508.233,A -85,B 0,C 180,E1 -18620.521,E2 -18620.521} C_VEL
LIN {X 0,Y 255.526,Z 510.497,A -85,B 0,C 180,E1 -18622.096,E2 -18622.096} C_VEL
LIN {X 0,Y 255.133,Z 512.336,A -85,B 0,C 180,E1 -18623.674,E2 -18623.674} C_VEL
LIN {X 0,Y 254.588,Z 514.704,A -85,B 0,C 180,E1 -18626.835,E2 -18626.835} C_VEL
LIN {X 0,Y 254.407,Z 515.537,A -85,B 0,C 180,E1 -18630,E2 -18630} C_VEL
LIN {X 0,Y 254.437,Z 515.345,A -85,B 0,C 180,E1 -18631.583,E2 -18631.583} C_VEL
LIN {X 0,Y 254.781,Z 513.802,A -85,B 0,C 180,E1 -18634.747,E2 -18634.747} C_VEL
LIN {X 0,Y 255.132,Z 512.452,A -85,B 0,C 180,E1 -18636.326,E2 -18636.326} C_VEL
LIN {X 0,Y 255.683,Z 509.714,A -85,B 0,C 180,E1 -18638.616,E2 -18638.616} C_VEL
LIN {X 0,Y 256.578,Z 505.747,A -85,B 0,C 180,E1 -18641.055,E2 -18641.055} C_VEL
LIN {X 0,Y 257.873,Z 500.753,A -85,B 0,C 180,E1 -18643.395,E2 -18643.395} C_VEL
LIN {X 0,Y 259.38,Z 494.464,A -85,B 0,C 180,E1 -18645.721,E2 -18645.721} C_VEL
LIN {X 0,Y 261.262,Z 486.586,A -85,B 0,C 180,E1 -18648.02,E2 -18648.02} C_VEL
LIN {X 0,Y 263.533,Z 476.775,A -85,B 0,C 180,E1 -18650.285,E2 -18650.285} C_VEL
LIN {X 0,Y 265.282,Z 466.926,A -85,B 0,C 180,E1 -18652.103,E2 -18652.103} C_VEL
LIN {X 0,Y 267.139,Z 456.299,A -85,B 0,C 180,E1 -18653.65,E2 -18653.65} C_VEL
LIN {X 0,Y 267.412,Z 453.446,A -85,B 0,C 180,E1 -18654.031,E2 -18654.031} C_VEL
LIN {X 0,Y 265.454,Z 442.773,A -85,B 0,C 180,E1 -18655.558,E2 -18655.558} C_VEL
LIN {X 0,Y 262.344,Z 431.094,A -85,B 0,C 180,E1 -18657.034,E2 -18657.034} C_VEL
LIN {X 0,Y 258.163,Z 419.01,A -85,B 0,C 180,E1 -18658.384,E2 -18658.384} C_VEL
LIN {X 0,Y 255.8,Z 413.139,A -85,B 0,C 180,E1 -18658.979,E2 -18658.979} C_VEL
LIN {X 0,Y 255.699,Z 412.588,A -85,B 0,C 180,E1 -18659.035,E2 -18659.035} C_VEL
LIN {X 0,Y 255.835,Z 410.784,A -85,B 0,C 180,E1 -18661.614,E2 -18661.614} C_VEL
LIN {X 0,Y 255.873,Z 408.832,A -85,B 0,C 180,E1 -18664.512,E2 -18664.512} C_VEL
LIN {X 0,Y 256.01,Z 408.596,A -85,B 0,C 180,E1 -18667.239,E2 -18667.239} C_VEL
LIN {X 0,Y 256.055,Z 408.589,A -85,B 0,C 180,E1 -18671.204,E2 -18671.204} C_VEL
LIN {X 0,Y 256.06,Z 408.586,A -85,B 0,C 180,E1 -18675.53,E2 -18675.53} C_VEL
LIN {X 0,Y 256.06,Z 408.589,A -85,B 0,C 180,E1 -18678.797,E2 -18678.797} C_VEL
LIN {X 0,Y 256.148,Z 408.577,A -85,B 0,C 180,E1 -18682.87,E2 -18682.87} C_VEL
LIN {X 0,Y 256.088,Z 408.585,A -85,B 0,C 180,E1 -18686.71,E2 -18686.71} C_VEL
LIN {X 0,Y 256.13,Z 408.579,A -85,B 0,C 180,E1 -18691.41,E2 -18691.41} C_VEL
LIN {X 0,Y 256.146,Z 408.577,A -85,B 0,C 180,E1 -18695.697,E2 -18695.697} C_VEL
LIN {X 0,Y 256.166,Z 408.574,A -85,B 0,C 180,E1 -18699.105,E2 -18699.105} C_VEL
LIN {X 0,Y 256.304,Z 408.56,A -85,B 0,C 180,E1 -18704.085,E2 -18704.085} C_VEL
LIN {X 0,Y 256.299,Z 408.558,A -85,B 0,C 180,E1 -18707.328,E2 -18707.328} C_VEL
LIN {X 0,Y 256.508,Z 408.533,A -85,B 0,C 180,E1 -18712.126,E2 -18712.126} C_VEL
LIN {X 0,Y 256.502,Z 408.535,A -85,B 0,C 180,E1 -18716.859,E2 -18716.859} C_VEL
LIN {X 0,Y 256.769,Z 408.503,A -85,B 0,C 180,E1 -18720,E2 -18720} C_VEL
LIN {X 0,Y 256.503,Z 408.536,A -85,B 0,C 180,E1 -18723.141,E2 -18723.141} C_VEL
LIN {X 0,Y 256.544,Z 408.531,A -85,B 0,C 180,E1 -18727.873,E2 -18727.873} C_VEL
LIN {X 0,Y 256.314,Z 408.559,A -85,B 0,C 180,E1 -18731.066,E2 -18731.066} C_VEL
LIN {X 0,Y 256.304,Z 408.557,A -85,B 0,C 180,E1 -18735.915,E2 -18735.915} C_VEL
LIN {X 0,Y 256.17,Z 408.573,A -85,B 0,C 180,E1 -18740.895,E2 -18740.895} C_VEL
LIN {X 0,Y 256.191,Z 408.574,A -85,B 0,C 180,E1 -18745.138,E2 -18745.138} C_VEL
LIN {X 0,Y 256.11,Z 408.582,A -85,B 0,C 180,E1 -18749.022,E2 -18749.022} C_VEL
LIN {X 0,Y 255.416,Z 408.677,A -85,B 0,C 180,E1 -18750.334,E2 -18750.334} C_VEL
LIN {X 0,Y 252.565,Z 409.034,A -85,B 0,C 180,E1 -18752.475,E2 -18752.475} C_VEL
LIN {X 0,Y 250.243,Z 409.779,A -85,B 0,C 180,E1 -18754.208,E2 -18754.208} C_VEL
LIN {X 0,Y 249.356,Z 410.681,A -85,B 0,C 180,E1 -18755.541,E2 -18755.541} C_VEL
LIN {X 0,Y 249.341,Z 411.058,A -85,B 0,C 180,E1 -18755.988,E2 -18755.988} C_VEL
LIN {X 0,Y 250.034,Z 414.98,A -85,B 0,C 180,E1 -18760.277,E2 -18760.277} C_VEL
LIN {X 0,Y 250.836,Z 419.161,A -85,B 0,C 180,E1 -18764.464,E2 -18764.464} C_VEL
LIN {X 0,Y 251.684,Z 423.999,A -85,B 0,C 180,E1 -18768.933,E2 -18768.933} C_VEL
LIN {X 0,Y 252.113,Z 427.755,A -85,B 0,C 180,E1 -18772.172,E2 -18772.172} C_VEL
LIN {X 0,Y 251.886,Z 430.169,A -85,B 0,C 180,E1 -18774.131,E2 -18774.131} C_VEL
LIN {X 0,Y 250.496,Z 436.065,A -85,B 0,C 180,E1 -18778.731,E2 -18778.731} C_VEL
LIN {X 0,Y 250.111,Z 438.027,A -85,B 0,C 180,E1 -18780.247,E2 -18780.247} C_VEL
LIN {X 0,Y 253.41,Z 452.279,A -85,B 0,C 180,E1 -18781.461,E2 -18781.461} C_VEL
LIN {X 0,Y 255.341,Z 463.521,A -85,B 0,C 180,E1 -18782.603,E2 -18782.603} C_VEL
LIN {X 0,Y 256.501,Z 473.369,A -85,B 0,C 180,E1 -18783.758,E2 -18783.758} C_VEL
LIN {X 0,Y 257.041,Z 484.791,A -85,B 0,C 180,E1 -18785.314,E2 -18785.314} C_VEL
LIN {X 0,Y 256.943,Z 495.59,A -85,B 0,C 180,E1 -18787.059,E2 -18787.059} C_VEL
LIN {X 0,Y 254.595,Z 506.089,A -85,B 0,C 180,E1 -18788.969,E2 -18788.969} C_VEL
LIN {X 0,Y 252.512,Z 515.413,A -85,B 0,C 180,E1 -18791.138,E2 -18791.138} C_VEL
LIN {X 0,Y 251.216,Z 521.69,A -85,B 0,C 180,E1 -18792.917,E2 -18792.917} C_VEL
LIN {X 0,Y 249.583,Z 528.628,A -85,B 0,C 180,E1 -18795.319,E2 -18795.319} C_VEL
LIN {X 0,Y 248.376,Z 534.2,A -85,B 0,C 180,E1 -18797.747,E2 -18797.747} C_VEL
LIN {X 0,Y 247.647,Z 538.586,A -85,B 0,C 180,E1 -18800.196,E2 -18800.196} C_VEL
LIN {X 0,Y 247.356,Z 540.915,A -85,B 0,C 180,E1 -18801.833,E2 -18801.833} C_VEL
LIN {X 0,Y 247.138,Z 543.706,A -85,B 0,C 180,E1 -18804.452,E2 -18804.452} C_VEL
LIN {X 0,Y 247.115,Z 545.244,A -85,B 0,C 180,E1 -18806.739,E2 -18806.739} C_VEL
LIN {X 0,Y 247.111,Z 545.864,A -85,B 0,C 180,E1 -18808.37,E2 -18808.37} C_VEL
LIN {X 0,Y 247.18,Z 546.085,A -85,B 0,C 180,E1 -18810,E2 -18810} C_VEL
LIN {X 0,Y 247.123,Z 545.858,A -85,B 0,C 180,E1 -18811.63,E2 -18811.63} C_VEL
LIN {X 0,Y 247.115,Z 545.234,A -85,B 0,C 180,E1 -18813.261,E2 -18813.261} C_VEL
LIN {X 0,Y 247.13,Z 543.705,A -85,B 0,C 180,E1 -18815.527,E2 -18815.527} C_VEL
LIN {X 0,Y 247.345,Z 540.885,A -85,B 0,C 180,E1 -18818.167,E2 -18818.167} C_VEL
LIN {X 0,Y 247.846,Z 537.214,A -85,B 0,C 180,E1 -18820.621,E2 -18820.621} C_VEL
LIN {X 0,Y 248.686,Z 532.43,A -85,B 0,C 180,E1 -18823.067,E2 -18823.067} C_VEL
LIN {X 0,Y 250.34,Z 525.275,A -85,B 0,C 180,E1 -18825.886,E2 -18825.886} C_VEL
LIN {X 0,Y 252.121,Z 517.682,A -85,B 0,C 180,E1 -18828.229,E2 -18828.229} C_VEL
LIN {X 0,Y 253.765,Z 509.573,A -85,B 0,C 180,E1 -18830.254,E2 -18830.254} C_VEL
LIN {X 0,Y 255.947,Z 499.913,A -85,B 0,C 180,E1 -18832.183,E2 -18832.183} C_VEL
LIN {X 0,Y 256.994,Z 494.244,A -85,B 0,C 180,E1 -18833.148,E2 -18833.148} C_VEL
LIN {X 0,Y 256.965,Z 482.692,A -85,B 0,C 180,E1 -18834.971,E2 -18834.971} C_VEL
LIN {X 0,Y 256.228,Z 471.036,A -85,B 0,C 180,E1 -18836.5,E2 -18836.5} C_VEL
LIN {X 0,Y 254.714,Z 459.527,A -85,B 0,C 180,E1 -18837.79,E2 -18837.79} C_VEL
LIN {X 0,Y 252.137,Z 446.53,A -85,B 0,C 180,E1 -18839.027,E2 -18839.027} C_VEL
LIN {X 0,Y 250.106,Z 438.01,A -85,B 0,C 180,E1 -18839.714,E2 -18839.714} C_VEL
LIN {X 0,Y 251.32,Z 432.494,A -85,B 0,C 180,E1 -18844.007,E2 -18844.007} C_VEL
LIN {X 0,Y 252.084,Z 428.922,A -85,B 0,C 180,E1 -18846.827,E2 -18846.827} C_VEL
LIN {X 0,Y 252.116,Z 426.675,A -85,B 0,C 180,E1 -18848.691,E2 -18848.691} C_VEL
LIN {X 0,Y 251.504,Z 422.772,A -85,B 0,C 180,E1 -18852.118,E2 -18852.118} C_VEL
LIN {X 0,Y 250.783,Z 419.131,A -85,B 0,C 180,E1 -18855.524,E2 -18855.524} C_VEL
LIN {X 0,Y 250.026,Z 414.93,A -85,B 0,C 180,E1 -18859.721,E2 -18859.721} C_VEL
LIN {X 0,Y 249.396,Z 411.205,A -85,B 0,C 180,E1 -18863.716,E2 -18863.716} C_VEL
LIN {X 0,Y 249.054,Z 409.462,A -85,B 0,C 180,E1 -18865.885,E2 -18865.885} C_VEL
LIN {X 0,Y 249.053,Z 409.461,A -85,B 0,C 180,E1 -18869.473,E2 -18869.473} C_VEL
LIN {X 0,Y 249.075,Z 409.46,A -85,B 0,C 180,E1 -18873.162,E2 -18873.162} C_VEL
LIN {X 0,Y 249.082,Z 409.46,A -85,B 0,C 180,E1 -18876.733,E2 -18876.733} C_VEL
LIN {X 0,Y 249.113,Z 409.455,A -85,B 0,C 180,E1 -18880.212,E2 -18880.212} C_VEL
LIN {X 0,Y 249.244,Z 409.438,A -85,B 0,C 180,E1 -18883.622,E2 -18883.622} C_VEL
LIN {X 0,Y 249.256,Z 409.439,A -85,B 0,C 180,E1 -18888.617,E2 -18888.617} C_VEL
LIN {X 0,Y 249.487,Z 409.408,A -85,B 0,C 180,E1 -18891.903,E2 -18891.903} C_VEL
LIN {X 0,Y 249.439,Z 409.414,A -85,B 0,C 180,E1 -18896.77,E2 -18896.77} C_VEL
LIN {X 0,Y 249.738,Z 409.376,A -85,B 0,C 180,E1 -18900,E2 -18900} C_VEL
LIN {X 0,Y 249.438,Z 409.412,A -85,B 0,C 180,E1 -18903.23,E2 -18903.23} C_VEL
LIN {X 0,Y 249.487,Z 409.408,A -85,B 0,C 180,E1 -18908.097,E2 -18908.097} C_VEL
LIN {X 0,Y 249.255,Z 409.435,A -85,B 0,C 180,E1 -18911.383,E2 -18911.383} C_VEL
LIN {X 0,Y 249.244,Z 409.439,A -85,B 0,C 180,E1 -18916.378,E2 -18916.378} C_VEL
LIN {X 0,Y 249.086,Z 409.457,A -85,B 0,C 180,E1 -18921.518,E2 -18921.518} C_VEL
LIN {X 0,Y 249.119,Z 409.453,A -85,B 0,C 180,E1 -18925.476,E2 -18925.476} C_VEL
LIN {X 0,Y 249.075,Z 409.457,A -85,B 0,C 180,E1 -18928.989,E2 -18928.989} C_VEL
LIN {X 0,Y 249.038,Z 409.458,A -85,B 0,C 180,E1 -18932.425,E2 -18932.425} C_VEL
LIN {X 0,Y 249.071,Z 409.455,A -85,B 0,C 180,E1 -18936.339,E2 -18936.339} C_VEL
LIN {X 0,Y 249.029,Z 409.463,A -85,B 0,C 180,E1 -18940.474,E2 -18940.474} C_VEL
LIN {X 0,Y 249.021,Z 409.465,A -85,B 0,C 180,E1 -18944.875,E2 -18944.875} C_VEL
LIN {X 0,Y 249.064,Z 409.462,A -85,B 0,C 180,E1 -18947.373,E2 -18947.373} C_VEL
LIN {X 0,Y 249.082,Z 409.459,A -85,B 0,C 180,E1 -18949.626,E2 -18949.626} C_VEL
LIN {X 0,Y 248.904,Z 409.486,A -85,B 0,C 180,E1 -18953.633,E2 -18953.633} C_VEL
LIN {X 0,Y 248.838,Z 409.587,A -85,B 0,C 180,E1 -18954.991,E2 -18954.991} C_VEL
LIN {X 0,Y 248.721,Z 412.532,A -85,B 0,C 180,E1 -18959.428,E2 -18959.428} C_VEL
LIN {X 0,Y 248.725,Z 413.054,A -85,B 0,C 180,E1 -18960.194,E2 -18960.194} C_VEL
LIN {X 0,Y 249.814,Z 416.231,A -85,B 0,C 180,E1 -18960.527,E2 -18960.527} C_VEL
LIN {X 0,Y 254.401,Z 428.166,A -85,B 0,C 180,E1 -18961.893,E2 -18961.893} C_VEL
LIN {X 0,Y 257.631,Z 439.089,A -85,B 0,C 180,E1 -18963.275,E2 -18963.275} C_VEL
LIN {X 0,Y 259.871,Z 449.05,A -85,B 0,C 180,E1 -18964.688,E2 -18964.688} C_VEL
LIN {X 0,Y 260.801,Z 454.984,A -85,B 0,C 180,E1 -18965.603,E2 -18965.603} C_VEL
LIN {X 0,Y 258.882,Z 466.455,A -85,B 0,C 180,E1 -18967.284,E2 -18967.284} C_VEL
LIN {X 0,Y 256.923,Z 476.655,A -85,B 0,C 180,E1 -18969.169,E2 -18969.169} C_VEL
LIN {X 0,Y 254.956,Z 485.105,A -85,B 0,C 180,E1 -18971.101,E2 -18971.101} C_VEL
LIN {X 0,Y 252.935,Z 493.313,A -85,B 0,C 180,E1 -18973.453,E2 -18973.453} C_VEL
LIN {X 0,Y 251.609,Z 498.916,A -85,B 0,C 180,E1 -18975.44,E2 -18975.44} C_VEL
LIN {X 0,Y 250.07,Z 504.387,A -85,B 0,C 180,E1 -18977.832,E2 -18977.832} C_VEL
LIN {X 0,Y 249.064,Z 508.665,A -85,B 0,C 180,E1 -18980.253,E2 -18980.253} C_VEL
LIN {X 0,Y 248.518,Z 510.929,A -85,B 0,C 180,E1 -18981.871,E2 -18981.871} C_VEL
LIN {X 0,Y 248.111,Z 512.768,A -85,B 0,C 180,E1 -18983.494,E2 -18983.494} C_VEL
LIN {X 0,Y 247.518,Z 515.135,A -85,B 0,C 180,E1 -18986.745,E2 -18986.745} C_VEL
LIN {X 0,Y 247.323,Z 515.969,A -85,B 0,C 180,E1 -18990,E2 -18990} C_VEL
LIN {X 0,Y 247.503,Z 515.193,A -85,B 0,C 180,E1 -18993.256,E2 -18993.256} C_VEL
LIN {X 0,Y 248.109,Z 512.882,A -85,B 0,C 180,E1 -18996.506,E2 -18996.506} C_VEL
LIN {X 0,Y 248.697,Z 510.04,A -85,B 0,C 180,E1 -18998.942,E2 -18998.942} C_VEL
LIN {X 0,Y 249.632,Z 506.177,A -85,B 0,C 180,E1 -19001.366,E2 -19001.366} C_VEL
LIN {X 0,Y 250.987,Z 501.183,A -85,B 0,C 180,E1 -19003.77,E2 -19003.77} C_VEL
LIN {X 0,Y 252.581,Z 494.893,A -85,B 0,C 180,E1 -19006.156,E2 -19006.156} C_VEL
LIN {X 0,Y 254.552,Z 487.014,A -85,B 0,C 180,E1 -19008.513,E2 -19008.513} C_VEL
LIN {X 0,Y 256.912,Z 477.202,A -85,B 0,C 180,E1 -19010.832,E2 -19010.832} C_VEL
LIN {X 0,Y 258.811,Z 466.91,A -85,B 0,C 180,E1 -19012.766,E2 -19012.766} C_VEL
LIN {X 0,Y 260.824,Z 455.604,A -85,B 0,C 180,E1 -19014.426,E2 -19014.426} C_VEL
LIN {X 0,Y 259.248,Z 445.931,A -85,B 0,C 180,E1 -19015.895,E2 -19015.895} C_VEL
LIN {X 0,Y 256.404,Z 434.496,A -85,B 0,C 180,E1 -19017.453,E2 -19017.453} C_VEL
LIN {X 0,Y 252.532,Z 422.8,A -85,B 0,C 180,E1 -19018.863,E2 -19018.863} C_VEL
LIN {X 0,Y 248.875,Z 413.734,A -85,B 0,C 180,E1 -19019.859,E2 -19019.859} C_VEL
LIN {X 0,Y 248.742,Z 413.013,A -85,B 0,C 180,E1 -19019.982,E2 -19019.982} C_VEL
LIN {X 0,Y 248.82,Z 411.336,A -85,B 0,C 180,E1 -19022.457,E2 -19022.457} C_VEL
LIN {X 0,Y 248.861,Z 409.67,A -85,B 0,C 180,E1 -19025.017,E2 -19025.017} C_VEL
LIN {X 0,Y 248.982,Z 409.472,A -85,B 0,C 180,E1 -19028.389,E2 -19028.389} C_VEL
LIN {X 0,Y 249.012,Z 409.466,A -85,B 0,C 180,E1 -19032.793,E2 -19032.793} C_VEL
LIN {X 0,Y 249.019,Z 409.465,A -85,B 0,C 180,E1 -19037.363,E2 -19037.363} C_VEL
LIN {X 0,Y 249.041,Z 409.46,A -85,B 0,C 180,E1 -19041.622,E2 -19041.622} C_VEL
LIN {X 0,Y 249.064,Z 409.457,A -85,B 0,C 180,E1 -19045.642,E2 -19045.642} C_VEL
LIN {X 0,Y 249.051,Z 409.461,A -85,B 0,C 180,E1 -19049.473,E2 -19049.473} C_VEL
LIN {X 0,Y 249.071,Z 409.458,A -85,B 0,C 180,E1 -19053.162,E2 -19053.162} C_VEL
LIN {X 0,Y 249.065,Z 409.459,A -85,B 0,C 180,E1 -19056.731,E2 -19056.731} C_VEL
LIN {X 0,Y 249.113,Z 409.454,A -85,B 0,C 180,E1 -19060.212,E2 -19060.212} C_VEL
LIN {X 0,Y 249.245,Z 409.437,A -85,B 0,C 180,E1 -19063.622,E2 -19063.622} C_VEL
LIN {X 0,Y 249.248,Z 409.436,A -85,B 0,C 180,E1 -19068.616,E2 -19068.616} C_VEL
LIN {X 0,Y 249.45,Z 409.413,A -85,B 0,C 180,E1 -19071.902,E2 -19071.902} C_VEL
LIN {X 0,Y 249.298,Z 409.431,A -85,B 0,C 180,E1 -19075.148,E2 -19075.148} C_VEL
LIN {X 0,Y 249.679,Z 409.385,A -85,B 0,C 180,E1 -19078.387,E2 -19078.387} C_VEL
LIN {X 0,Y 249.68,Z 409.387,A -85,B 0,C 180,E1 -19081.613,E2 -19081.613} C_VEL
LIN {X 0,Y 249.466,Z 409.409,A -85,B 0,C 180,E1 -19086.47,E2 -19086.47} C_VEL
LIN {X 0,Y 249.428,Z 409.417,A -85,B 0,C 180,E1 -19089.733,E2 -19089.733} C_VEL
LIN {X 0,Y 249.21,Z 409.441,A -85,B 0,C 180,E1 -19094.703,E2 -19094.703} C_VEL
LIN {X 0,Y 249.143,Z 409.447,A -85,B 0,C 180,E1 -19098.077,E2 -19098.077} C_VEL
LIN {X 0,Y 249.091,Z 409.454,A -85,B 0,C 180,E1 -19101.518,E2 -19101.518} C_VEL
LIN {X 0,Y 249.134,Z 409.453,A -85,B 0,C 180,E1 -19105.482,E2 -19105.482} C_VEL
LIN {X 0,Y 249.076,Z 409.461,A -85,B 0,C 180,E1 -19108.994,E2 -19108.994} C_VEL
LIN {X 0,Y 249.04,Z 409.465,A -85,B 0,C 180,E1 -19113.873,E2 -19113.873} C_VEL
LIN {X 0,Y 249.232,Z 410.301,A -85,B 0,C 180,E1 -19115.138,E2 -19115.138} C_VEL
LIN {X 0,Y 249.341,Z 411.058,A -85,B 0,C 180,E1 -19115.988,E2 -19115.988} C_VEL
LIN {X 0,Y 248.911,Z 412.379,A -85,B 0,C 180,E1 -19117.304,E2 -19117.304} C_VEL
LIN {X 0,Y 246.483,Z 414.921,A -85,B 0,C 180,E1 -19119.444,E2 -19119.444} C_VEL
LIN {X 0,Y 244.394,Z 417.034,A -85,B 0,C 180,E1 -19121.181,E2 -19121.181} C_VEL
LIN {X 0,Y 243.585,Z 418.521,A -85,B 0,C 180,E1 -19122.525,E2 -19122.525} C_VEL
LIN {X 0,Y 243.571,Z 418.981,A -85,B 0,C 180,E1 -19122.98,E2 -19122.98} C_VEL
LIN {X 0,Y 244.368,Z 423.345,A -85,B 0,C 180,E1 -19127.235,E2 -19127.235} C_VEL
LIN {X 0,Y 245.042,Z 427.298,A -85,B 0,C 180,E1 -19130.877,E2 -19130.877} C_VEL
LIN {X 0,Y 244.965,Z 430.305,A -85,B 0,C 180,E1 -19133.448,E2 -19133.448} C_VEL
LIN {X 0,Y 243.98,Z 434.449,A -85,B 0,C 180,E1 -19136.817,E2 -19136.817} C_VEL
LIN {X 0,Y 243.272,Z 437.571,A -85,B 0,C 180,E1 -19139.323,E2 -19139.323} C_VEL
LIN {X 0,Y 246.698,Z 452.09,A -85,B 0,C 180,E1 -19140.63,E2 -19140.63} C_VEL
LIN {X 0,Y 248.788,Z 464.302,A -85,B 0,C 180,E1 -19141.941,E2 -19141.941} C_VEL
LIN {X 0,Y 249.992,Z 476.057,A -85,B 0,C 180,E1 -19143.414,E2 -19143.414} C_VEL
LIN {X 0,Y 250.361,Z 487.524,A -85,B 0,C 180,E1 -19145.097,E2 -19145.097} C_VEL
LIN {X 0,Y 250.154,Z 496.34,A -85,B 0,C 180,E1 -19146.619,E2 -19146.619} C_VEL
LIN {X 0,Y 247.959,Z 505.658,A -85,B 0,C 180,E1 -19148.379,E2 -19148.379} C_VEL
LIN {X 0,Y 245.817,Z 514.773,A -85,B 0,C 180,E1 -19150.544,E2 -19150.544} C_VEL
LIN {X 0,Y 244.066,Z 522.5,A -85,B 0,C 180,E1 -19152.833,E2 -19152.833} C_VEL
LIN {X 0,Y 242.461,Z 529.217,A -85,B 0,C 180,E1 -19155.307,E2 -19155.307} C_VEL
LIN {X 0,Y 241.123,Z 535.377,A -85,B 0,C 180,E1 -19158.227,E2 -19158.227} C_VEL
LIN {X 0,Y 240.441,Z 539.393,A -85,B 0,C 180,E1 -19160.749,E2 -19160.749} C_VEL
LIN {X 0,Y 240.087,Z 542.371,A -85,B 0,C 180,E1 -19163.276,E2 -19163.276} C_VEL
LIN {X 0,Y 240.009,Z 543.793,A -85,B 0,C 180,E1 -19164.96,E2 -19164.96} C_VEL
LIN {X 0,Y 240.027,Z 544.812,A -85,B 0,C 180,E1 -19166.643,E2 -19166.643} C_VEL
LIN {X 0,Y 240.038,Z 545.433,A -85,B 0,C 180,E1 -19168.322,E2 -19168.322} C_VEL
LIN {X 0,Y 240.102,Z 545.654,A -85,B 0,C 180,E1 -19170,E2 -19170} C_VEL
LIN {X 0,Y 240.05,Z 545.427,A -85,B 0,C 180,E1 -19171.678,E2 -19171.678} C_VEL
LIN {X 0,Y 240.027,Z 544.801,A -85,B 0,C 180,E1 -19173.357,E2 -19173.357} C_VEL
LIN {X 0,Y 240.027,Z 543.504,A -85,B 0,C 180,E1 -19175.423,E2 -19175.423} C_VEL
LIN {X 0,Y 240.296,Z 540.45,A -85,B 0,C 180,E1 -19178.409,E2 -19178.409} C_VEL
LIN {X 0,Y 240.842,Z 536.778,A -85,B 0,C 180,E1 -19180.934,E2 -19180.934} C_VEL
LIN {X 0,Y 241.734,Z 531.993,A -85,B 0,C 180,E1 -19183.449,E2 -19183.449} C_VEL
LIN {X 0,Y 243.233,Z 525.969,A -85,B 0,C 180,E1 -19185.932,E2 -19185.932} C_VEL
LIN {X 0,Y 245.055,Z 518.472,A -85,B 0,C 180,E1 -19188.389,E2 -19188.389} C_VEL
LIN {X 0,Y 246.686,Z 510.829,A -85,B 0,C 180,E1 -19190.426,E2 -19190.426} C_VEL
LIN {X 0,Y 248.909,Z 501.607,A -85,B 0,C 180,E1 -19192.406,E2 -19192.406} C_VEL
LIN {X 0,Y 250.212,Z 494.987,A -85,B 0,C 180,E1 -19193.594,E2 -19193.594} C_VEL
LIN {X 0,Y 250.277,Z 483.482,A -85,B 0,C 180,E1 -19195.501,E2 -19195.501} C_VEL
LIN {X 0,Y 249.595,Z 471.074,A -85,B 0,C 180,E1 -19197.206,E2 -19197.206} C_VEL
LIN {X 0,Y 248.07,Z 459.455,A -85,B 0,C 180,E1 -19198.567,E2 -19198.567} C_VEL
LIN {X 0,Y 245.385,Z 446.316,A -85,B 0,C 180,E1 -19199.889,E2 -19199.889} C_VEL
LIN {X 0,Y 243.27,Z 437.479,A -85,B 0,C 180,E1 -19200.677,E2 -19200.677} C_VEL
LIN {X 0,Y 244.592,Z 432.052,A -85,B 0,C 180,E1 -19205.077,E2 -19205.077} C_VEL
LIN {X 0,Y 245.067,Z 429.673,A -85,B 0,C 180,E1 -19207.03,E2 -19207.03} C_VEL
LIN {X 0,Y 244.864,Z 426.019,A -85,B 0,C 180,E1 -19210.224,E2 -19210.224} C_VEL
LIN {X 0,Y 244.137,Z 421.991,A -85,B 0,C 180,E1 -19213.972,E2 -19213.972} C_VEL
LIN {X 0,Y 243.253,Z 417.309,A -85,B 0,C 180,E1 -19218.693,E2 -19218.693} C_VEL
LIN {X 0,Y 242.599,Z 413.748,A -85,B 0,C 180,E1 -19222.529,E2 -19222.529} C_VEL
LIN {X 0,Y 242.012,Z 410.339,A -85,B 0,C 180,E1 -19226.767,E2 -19226.767} C_VEL
LIN {X 0,Y 242.038,Z 410.337,A -85,B 0,C 180,E1 -19230.587,E2 -19230.587} C_VEL
LIN {X 0,Y 242.069,Z 410.332,A -85,B 0,C 180,E1 -19234.183,E2 -19234.183} C_VEL
LIN {X 0,Y 242.055,Z 410.335,A -85,B 0,C 180,E1 -19238.297,E2 -19238.297} C_VEL
LIN {X 0,Y 242.165,Z 410.32,A -85,B 0,C 180,E1 -19243.278,E2 -19243.278} C_VEL
LIN {X 0,Y 242.19,Z 410.319,A -85,B 0,C 180,E1 -19248.28,E2 -19248.28} C_VEL
LIN {X 0,Y 242.438,Z 410.285,A -85,B 0,C 180,E1 -19251.666,E2 -19251.666} C_VEL
LIN {X 0,Y 242.263,Z 410.308,A -85,B 0,C 180,E1 -19255.007,E2 -19255.007} C_VEL
LIN {X 0,Y 242.639,Z 410.262,A -85,B 0,C 180,E1 -19258.34,E2 -19258.34} C_VEL
LIN {X 0,Y 242.639,Z 410.259,A -85,B 0,C 180,E1 -19261.66,E2 -19261.66} C_VEL
LIN {X 0,Y 242.432,Z 410.284,A -85,B 0,C 180,E1 -19266.75,E2 -19266.75} C_VEL
LIN {X 0,Y 242.348,Z 410.297,A -85,B 0,C 180,E1 -19270.02,E2 -19270.02} C_VEL
LIN {X 0,Y 242.17,Z 410.318,A -85,B 0,C 180,E1 -19275.141,E2 -19275.141} C_VEL
LIN {X 0,Y 242.075,Z 410.329,A -85,B 0,C 180,E1 -19278.624,E2 -19278.624} C_VEL
LIN {X 0,Y 242.009,Z 410.34,A -85,B 0,C 180,E1 -19282.181,E2 -19282.181} C_VEL
LIN {X 0,Y 242.068,Z 410.333,A -85,B 0,C 180,E1 -19285.838,E2 -19285.838} C_VEL
LIN {X 0,Y 242.009,Z 410.339,A -85,B 0,C 180,E1 -19289.583,E2 -19289.583} C_VEL
LIN {X 0,Y 241.993,Z 410.337,A -85,B 0,C 180,E1 -19293.491,E2 -19293.491} C_VEL
LIN {X 0,Y 242.004,Z 410.337,A -85,B 0,C 180,E1 -19297.579,E2 -19297.579} C_VEL
LIN {X 0,Y 241.95,Z 410.347,A -85,B 0,C 180,E1 -19301.92,E2 -19301.92} C_VEL
LIN {X 0,Y 241.993,Z 410.341,A -85,B 0,C 180,E1 -19306.557,E2 -19306.557} C_VEL
LIN {X 0,Y 241.999,Z 410.343,A -85,B 0,C 180,E1 -19310.289,E2 -19310.289} C_VEL
LIN {X 0,Y 241.83,Z 410.448,A -85,B 0,C 180,E1 -19314.462,E2 -19314.462} C_VEL
LIN {X 0,Y 241.728,Z 413.523,A -85,B 0,C 180,E1 -19319.202,E2 -19319.202} C_VEL
LIN {X 0,Y 241.901,Z 414.43,A -85,B 0,C 180,E1 -19319.335,E2 -19319.335} C_VEL
LIN {X 0,Y 246.862,Z 426.675,A -85,B 0,C 180,E1 -19320.797,E2 -19320.797} C_VEL
LIN {X 0,Y 250.21,Z 437.253,A -85,B 0,C 180,E1 -19322.176,E2 -19322.176} C_VEL
LIN {X 0,Y 252.848,Z 448.205,A -85,B 0,C 180,E1 -19323.764,E2 -19323.764} C_VEL
LIN {X 0,Y 254.231,Z 456.841,A -85,B 0,C 180,E1 -19325.149,E2 -19325.149} C_VEL
LIN {X 0,Y 252.364,Z 466.89,A -85,B 0,C 180,E1 -19326.663,E2 -19326.663} C_VEL
LIN {X 0,Y 250.327,Z 477.089,A -85,B 0,C 180,E1 -19328.594,E2 -19328.594} C_VEL
LIN {X 0,Y 248.275,Z 485.539,A -85,B 0,C 180,E1 -19330.573,E2 -19330.573} C_VEL
LIN {X 0,Y 246.501,Z 492.525,A -85,B 0,C 180,E1 -19332.581,E2 -19332.581} C_VEL
LIN {X 0,Y 244.754,Z 499.349,A -85,B 0,C 180,E1 -19335.023,E2 -19335.023} C_VEL
LIN {X 0,Y 243.159,Z 504.819,A -85,B 0,C 180,E1 -19337.481,E2 -19337.481} C_VEL
LIN {X 0,Y 242.07,Z 509.099,A -85,B 0,C 180,E1 -19339.968,E2 -19339.968} C_VEL
LIN {X 0,Y 241.463,Z 511.486,A -85,B 0,C 180,E1 -19341.732,E2 -19341.732} C_VEL
LIN {X 0,Y 241.068,Z 513.2,A -85,B 0,C 180,E1 -19343.303,E2 -19343.303} C_VEL
LIN {X 0,Y 240.698,Z 514.584,A -85,B 0,C 180,E1 -19344.975,E2 -19344.975} C_VEL
LIN {X 0,Y 240.282,Z 516.173,A -85,B 0,C 180,E1 -19348.324,E2 -19348.324} C_VEL
LIN {X 0,Y 240.241,Z 516.4,A -85,B 0,C 180,E1 -19350,E2 -19350} C_VEL
LIN {X 0,Y 240.437,Z 515.624,A -85,B 0,C 180,E1 -19353.352,E2 -19353.352} C_VEL
LIN {X 0,Y 241.063,Z 513.313,A -85,B 0,C 180,E1 -19356.697,E2 -19356.697} C_VEL
LIN {X 0,Y 241.708,Z 510.47,A -85,B 0,C 180,E1 -19359.202,E2 -19359.202} C_VEL
LIN {X 0,Y 242.705,Z 506.607,A -85,B 0,C 180,E1 -19361.695,E2 -19361.695} C_VEL
LIN {X 0,Y 244.114,Z 501.613,A -85,B 0,C 180,E1 -19364.165,E2 -19364.165} C_VEL
LIN {X 0,Y 245.779,Z 495.322,A -85,B 0,C 180,E1 -19366.616,E2 -19366.616} C_VEL
LIN {X 0,Y 247.856,Z 487.442,A -85,B 0,C 180,E1 -19369.032,E2 -19369.032} C_VEL
LIN {X 0,Y 250.314,Z 477.63,A -85,B 0,C 180,E1 -19371.408,E2 -19371.408} C_VEL
LIN {X 0,Y 252.299,Z 467.337,A -85,B 0,C 180,E1 -19373.388,E2 -19373.388} C_VEL
LIN {X 0,Y 254.155,Z 457.526,A -85,B 0,C 180,E1 -19374.88,E2 -19374.88} C_VEL
LIN {X 0,Y 253.632,Z 452.508,A -85,B 0,C 180,E1 -19375.688,E2 -19375.688} C_VEL
LIN {X 0,Y 251.689,Z 442.863,A -85,B 0,C 180,E1 -19377.161,E2 -19377.161} C_VEL
LIN {X 0,Y 248.479,Z 431.335,A -85,B 0,C 180,E1 -19378.74,E2 -19378.74} C_VEL
LIN {X 0,Y 244.167,Z 419.716,A -85,B 0,C 180,E1 -19380.19,E2 -19380.19} C_VEL
LIN {X 0,Y 241.804,Z 413.823,A -85,B 0,C 180,E1 -19380.846,E2 -19380.846} C_VEL
LIN {X 0,Y 241.734,Z 413.475,A -85,B 0,C 180,E1 -19380.949,E2 -19380.949} C_VEL
LIN {X 0,Y 241.814,Z 411.79,A -85,B 0,C 180,E1 -19383.519,E2 -19383.519} C_VEL
LIN {X 0,Y 241.83,Z 410.536,A -85,B 0,C 180,E1 -19385.538,E2 -19385.538} C_VEL
LIN {X 0,Y 241.952,Z 410.347,A -85,B 0,C 180,E1 -19388.346,E2 -19388.346} C_VEL
LIN {X 0,Y 241.935,Z 410.348,A -85,B 0,C 180,E1 -19391.923,E2 -19391.923} C_VEL
LIN {X 0,Y 241.937,Z 410.35,A -85,B 0,C 180,E1 -19396.571,E2 -19396.571} C_VEL
LIN {X 0,Y 241.975,Z 410.342,A -85,B 0,C 180,E1 -19400.284,E2 -19400.284} C_VEL
LIN {X 0,Y 242.04,Z 410.332,A -85,B 0,C 180,E1 -19404.498,E2 -19404.498} C_VEL
LIN {X 0,Y 241.978,Z 410.344,A -85,B 0,C 180,E1 -19408.48,E2 -19408.48} C_VEL
LIN {X 0,Y 242.004,Z 410.34,A -85,B 0,C 180,E1 -19412.312,E2 -19412.312} C_VEL
LIN {X 0,Y 242.045,Z 410.336,A -85,B 0,C 180,E1 -19416.014,E2 -19416.014} C_VEL
LIN {X 0,Y 242.039,Z 410.336,A -85,B 0,C 180,E1 -19419.608,E2 -19419.608} C_VEL
LIN {X 0,Y 242.167,Z 410.318,A -85,B 0,C 180,E1 -19423.278,E2 -19423.278} C_VEL
LIN {X 0,Y 242.185,Z 410.317,A -85,B 0,C 180,E1 -19428.28,E2 -19428.28} C_VEL
LIN {X 0,Y 242.398,Z 410.293,A -85,B 0,C 180,E1 -19431.664,E2 -19431.664} C_VEL
LIN {X 0,Y 242.258,Z 410.308,A -85,B 0,C 180,E1 -19435.007,E2 -19435.007} C_VEL
LIN {X 0,Y 242.64,Z 410.262,A -85,B 0,C 180,E1 -19438.34,E2 -19438.34} C_VEL
LIN {X 0,Y 242.64,Z 410.264,A -85,B 0,C 180,E1 -19441.66,E2 -19441.66} C_VEL
LIN {X 0,Y 242.438,Z 410.285,A -85,B 0,C 180,E1 -19446.659,E2 -19446.659} C_VEL
LIN {X 0,Y 242.349,Z 410.298,A -85,B 0,C 180,E1 -19450.02,E2 -19450.02} C_VEL
LIN {X 0,Y 242.171,Z 410.32,A -85,B 0,C 180,E1 -19455.141,E2 -19455.141} C_VEL
LIN {X 0,Y 242.077,Z 410.328,A -85,B 0,C 180,E1 -19458.624,E2 -19458.624} C_VEL
LIN {X 0,Y 242.016,Z 410.338,A -85,B 0,C 180,E1 -19462.18,E2 -19462.18} C_VEL
LIN {X 0,Y 242.069,Z 410.333,A -85,B 0,C 180,E1 -19465.838,E2 -19465.838} C_VEL
LIN {X 0,Y 242.01,Z 410.34,A -85,B 0,C 180,E1 -19469.583,E2 -19469.583} C_VEL
LIN {X 0,Y 242.036,Z 410.506,A -85,B 0,C 180,E1 -19473.484,E2 -19473.484} C_VEL
LIN {X 0,Y 242.622,Z 413.851,A -85,B 0,C 180,E1 -19477.467,E2 -19477.467} C_VEL
LIN {X 0,Y 243.534,Z 418.706,A -85,B 0,C 180,E1 -19482.701,E2 -19482.701} C_VEL
LIN {X 0,Y 243.571,Z 418.981,A -85,B 0,C 180,E1 -19482.98,E2 -19482.98} C_VEL
LIN {X 0,Y 243.123,Z 420.453,A -85,B 0,C 180,E1 -19484.323,E2 -19484.323} C_VEL
LIN {X 0,Y 240.689,Z 423.187,A -85,B 0,C 180,E1 -19486.507,E2 -19486.507} C_VEL
LIN {X 0,Y 238.636,Z 425.432,A -85,B 0,C 180,E1 -19488.28,E2 -19488.28} C_VEL
LIN {X 0,Y 237.888,Z 427.04,A -85,B 0,C 180,E1 -19489.652,E2 -19489.652} C_VEL
LIN {X 0,Y 237.901,Z 427.546,A -85,B 0,C 180,E1 -19490.116,E2 -19490.116} C_VEL
LIN {X 0,Y 238.022,Z 430.595,A -85,B 0,C 180,E1 -19492.866,E2 -19492.866} C_VEL
LIN {X 0,Y 237.121,Z 434.409,A -85,B 0,C 180,E1 -19496.087,E2 -19496.087} C_VEL
LIN {X 0,Y 236.442,Z 437.129,A -85,B 0,C 180,E1 -19498.35,E2 -19498.35} C_VEL
LIN {X 0,Y 238.024,Z 443.372,A -85,B 0,C 180,E1 -19498.9,E2 -19498.9} C_VEL
LIN {X 0,Y 240.69,Z 455.069,A -85,B 0,C 180,E1 -19500.088,E2 -19500.088} C_VEL
LIN {X 0,Y 242.406,Z 466.309,A -85,B 0,C 180,E1 -19501.387,E2 -19501.387} C_VEL
LIN {X 0,Y 243.427,Z 477.139,A -85,B 0,C 180,E1 -19502.838,E2 -19502.838} C_VEL
LIN {X 0,Y 243.653,Z 488.408,A -85,B 0,C 180,E1 -19504.592,E2 -19504.592} C_VEL
LIN {X 0,Y 243.387,Z 497.045,A -85,B 0,C 180,E1 -19506.155,E2 -19506.155} C_VEL
LIN {X 0,Y 240.873,Z 507.029,A -85,B 0,C 180,E1 -19508.16,E2 -19508.16} C_VEL
LIN {X 0,Y 238.641,Z 516.095,A -85,B 0,C 180,E1 -19510.46,E2 -19510.46} C_VEL
LIN {X 0,Y 237.279,Z 522.069,A -85,B 0,C 180,E1 -19512.326,E2 -19512.326} C_VEL
LIN {X 0,Y 235.546,Z 528.783,A -85,B 0,C 180,E1 -19514.866,E2 -19514.866} C_VEL
LIN {X 0,Y 234.131,Z 534.942,A -85,B 0,C 180,E1 -19517.87,E2 -19517.87} C_VEL
LIN {X 0,Y 233.409,Z 538.96,A -85,B 0,C 180,E1 -19520.467,E2 -19520.467} C_VEL
LIN {X 0,Y 233.012,Z 541.937,A -85,B 0,C 180,E1 -19523.07,E2 -19523.07} C_VEL
LIN {X 0,Y 232.925,Z 543.36,A -85,B 0,C 180,E1 -19524.806,E2 -19524.806} C_VEL
LIN {X 0,Y 232.942,Z 544.38,A -85,B 0,C 180,E1 -19526.54,E2 -19526.54} C_VEL
LIN {X 0,Y 232.967,Z 545.002,A -85,B 0,C 180,E1 -19528.271,E2 -19528.271} C_VEL
LIN {X 0,Y 233.026,Z 545.223,A -85,B 0,C 180,E1 -19530,E2 -19530} C_VEL
LIN {X 0,Y 232.977,Z 544.995,A -85,B 0,C 180,E1 -19531.728,E2 -19531.728} C_VEL
LIN {X 0,Y 232.942,Z 544.368,A -85,B 0,C 180,E1 -19533.459,E2 -19533.459} C_VEL
LIN {X 0,Y 232.954,Z 543.216,A -85,B 0,C 180,E1 -19535.388,E2 -19535.388} C_VEL
LIN {X 0,Y 233.244,Z 540.015,A -85,B 0,C 180,E1 -19538.665,E2 -19538.665} C_VEL
LIN {X 0,Y 233.854,Z 536.344,A -85,B 0,C 180,E1 -19541.265,E2 -19541.265} C_VEL
LIN {X 0,Y 234.803,Z 531.558,A -85,B 0,C 180,E1 -19543.854,E2 -19543.854} C_VEL
LIN {X 0,Y 236.34,Z 525.53,A -85,B 0,C 180,E1 -19546.409,E2 -19546.409} C_VEL
LIN {X 0,Y 238.267,Z 518.034,A -85,B 0,C 180,E1 -19548.933,E2 -19548.933} C_VEL
LIN {X 0,Y 239.996,Z 510.391,A -85,B 0,C 180,E1 -19551.022,E2 -19551.022} C_VEL
LIN {X 0,Y 242.33,Z 501.169,A -85,B 0,C 180,E1 -19553.049,E2 -19553.049} C_VEL
LIN {X 0,Y 243.443,Z 495.729,A -85,B 0,C 180,E1 -19554.065,E2 -19554.065} C_VEL
LIN {X 0,Y 243.615,Z 484.22,A -85,B 0,C 180,E1 -19556.062,E2 -19556.062} C_VEL
LIN {X 0,Y 243.095,Z 472.687,A -85,B 0,C 180,E1 -19557.746,E2 -19557.746} C_VEL
LIN {X 0,Y 241.644,Z 460.69,A -85,B 0,C 180,E1 -19559.247,E2 -19559.247} C_VEL
LIN {X 0,Y 239.002,Z 447.396,A -85,B 0,C 180,E1 -19560.67,E2 -19560.67} C_VEL
LIN {X 0,Y 236.452,Z 437.042,A -85,B 0,C 180,E1 -19561.651,E2 -19561.651} C_VEL
LIN {X 0,Y 237.578,Z 432.761,A -85,B 0,C 180,E1 -19565.229,E2 -19565.229} C_VEL
LIN {X 0,Y 238.034,Z 430.545,A -85,B 0,C 180,E1 -19567.138,E2 -19567.138} C_VEL
LIN {X 0,Y 237.921,Z 427.539,A -85,B 0,C 180,E1 -19569.823,E2 -19569.823} C_VEL
LIN {X 0,Y 237.334,Z 424.298,A -85,B 0,C 180,E1 -19572.928,E2 -19572.928} C_VEL
LIN {X 0,Y 236.584,Z 420.353,A -85,B 0,C 180,E1 -19576.903,E2 -19576.903} C_VEL
LIN {X 0,Y 235.818,Z 416.357,A -85,B 0,C 180,E1 -19581.255,E2 -19581.255} C_VEL
LIN {X 0,Y 235.248,Z 412.889,A -85,B 0,C 180,E1 -19585.415,E2 -19585.415} C_VEL
LIN {X 0,Y 234.955,Z 411.222,A -85,B 0,C 180,E1 -19587.678,E2 -19587.678} C_VEL
LIN {X 0,Y 234.953,Z 411.219,A -85,B 0,C 180,E1 -19591.406,E2 -19591.406} C_VEL
LIN {X 0,Y 234.989,Z 411.213,A -85,B 0,C 180,E1 -19595.247,E2 -19595.247} C_VEL
LIN {X 0,Y 235.014,Z 411.211,A -85,B 0,C 180,E1 -19598.97,E2 -19598.97} C_VEL
LIN {X 0,Y 235.098,Z 411.201,A -85,B 0,C 180,E1 -19603.059,E2 -19603.059} C_VEL
LIN {X 0,Y 235.15,Z 411.195,A -85,B 0,C 180,E1 -19607.924,E2 -19607.924} C_VEL
LIN {X 0,Y 235.393,Z 411.163,A -85,B 0,C 180,E1 -19611.415,E2 -19611.415} C_VEL
LIN {X 0,Y 235.408,Z 411.162,A -85,B 0,C 180,E1 -19613.142,E2 -19613.142} C_VEL
LIN {X 0,Y 235.599,Z 411.139,A -85,B 0,C 180,E1 -19618.291,E2 -19618.291} C_VEL
LIN {X 0,Y 235.599,Z 411.136,A -85,B 0,C 180,E1 -19621.709,E2 -19621.709} C_VEL
LIN {X 0,Y 235.409,Z 411.159,A -85,B 0,C 180,E1 -19626.859,E2 -19626.859} C_VEL
LIN {X 0,Y 235.256,Z 411.18,A -85,B 0,C 180,E1 -19630.326,E2 -19630.326} C_VEL
LIN {X 0,Y 235.116,Z 411.197,A -85,B 0,C 180,E1 -19635.606,E2 -19635.606} C_VEL
LIN {X 0,Y 235.01,Z 411.208,A -85,B 0,C 180,E1 -19639.206,E2 -19639.206} C_VEL
LIN {X 0,Y 234.955,Z 411.217,A -85,B 0,C 180,E1 -19642.884,E2 -19642.884} C_VEL
LIN {X 0,Y 234.969,Z 411.214,A -85,B 0,C 180,E1 -19646.658,E2 -19646.658} C_VEL
LIN {X 0,Y 234.925,Z 411.221,A -85,B 0,C 180,E1 -19650.569,E2 -19650.569} C_VEL
LIN {X 0,Y 234.963,Z 411.216,A -85,B 0,C 180,E1 -19654.633,E2 -19654.633} C_VEL
LIN {X 0,Y 234.943,Z 411.219,A -85,B 0,C 180,E1 -19658.944,E2 -19658.944} C_VEL
LIN {X 0,Y 234.924,Z 411.22,A -85,B 0,C 180,E1 -19663.478,E2 -19663.478} C_VEL
LIN {X 0,Y 234.967,Z 411.216,A -85,B 0,C 180,E1 -19666.532,E2 -19666.532} C_VEL
LIN {X 0,Y 234.941,Z 411.222,A -85,B 0,C 180,E1 -19671.083,E2 -19671.083} C_VEL
LIN {X 0,Y 234.796,Z 411.338,A -85,B 0,C 180,E1 -19673.918,E2 -19673.918} C_VEL
LIN {X 0,Y 234.768,Z 414.13,A -85,B 0,C 180,E1 -19678.254,E2 -19678.254} C_VEL
LIN {X 0,Y 235.941,Z 417.266,A -85,B 0,C 180,E1 -19678.606,E2 -19678.606} C_VEL
LIN {X 0,Y 240.497,Z 428.577,A -85,B 0,C 180,E1 -19680.062,E2 -19680.062} C_VEL
LIN {X 0,Y 244.018,Z 439.847,A -85,B 0,C 180,E1 -19681.633,E2 -19681.633} C_VEL
LIN {X 0,Y 246.528,Z 450.828,A -85,B 0,C 180,E1 -19683.33,E2 -19683.33} C_VEL
LIN {X 0,Y 247.623,Z 458.514,A -85,B 0,C 180,E1 -19684.636,E2 -19684.636} C_VEL
LIN {X 0,Y 245.479,Z 469.404,A -85,B 0,C 180,E1 -19686.371,E2 -19686.371} C_VEL
LIN {X 0,Y 243.291,Z 479.322,A -85,B 0,C 180,E1 -19688.389,E2 -19688.389} C_VEL
LIN {X 0,Y 240.815,Z 488.918,A -85,B 0,C 180,E1 -19690.833,E2 -19690.833} C_VEL
LIN {X 0,Y 238.748,Z 496.559,A -85,B 0,C 180,E1 -19693.321,E2 -19693.321} C_VEL
LIN {X 0,Y 237.311,Z 501.772,A -85,B 0,C 180,E1 -19695.42,E2 -19695.42} C_VEL
LIN {X 0,Y 235.82,Z 506.827,A -85,B 0,C 180,E1 -19697.959,E2 -19697.959} C_VEL
LIN {X 0,Y 234.79,Z 510.742,A -85,B 0,C 180,E1 -19700.524,E2 -19700.524} C_VEL
LIN {X 0,Y 234.03,Z 513.632,A -85,B 0,C 180,E1 -19703.101,E2 -19703.101} C_VEL
LIN {X 0,Y 233.657,Z 515.015,A -85,B 0,C 180,E1 -19704.823,E2 -19704.823} C_VEL
LIN {X 0,Y 233.207,Z 516.604,A -85,B 0,C 180,E1 -19708.273,E2 -19708.273} C_VEL
LIN {X 0,Y 233.161,Z 516.831,A -85,B 0,C 180,E1 -19710,E2 -19710} C_VEL
LIN {X 0,Y 233.374,Z 516.055,A -85,B 0,C 180,E1 -19713.453,E2 -19713.453} C_VEL
LIN {X 0,Y 234.024,Z 513.744,A -85,B 0,C 180,E1 -19716.9,E2 -19716.9} C_VEL
LIN {X 0,Y 234.703,Z 510.902,A -85,B 0,C 180,E1 -19719.48,E2 -19719.48} C_VEL
LIN {X 0,Y 235.765,Z 507.037,A -85,B 0,C 180,E1 -19722.044,E2 -19722.044} C_VEL
LIN {X 0,Y 237.255,Z 502.042,A -85,B 0,C 180,E1 -19724.584,E2 -19724.584} C_VEL
LIN {X 0,Y 239.006,Z 495.751,A -85,B 0,C 180,E1 -19727.101,E2 -19727.101} C_VEL
LIN {X 0,Y 241.173,Z 487.87,A -85,B 0,C 180,E1 -19729.58,E2 -19729.58} C_VEL
LIN {X 0,Y 243.742,Z 478.057,A -85,B 0,C 180,E1 -19732.015,E2 -19732.015} C_VEL
LIN {X 0,Y 245.817,Z 467.764,A -85,B 0,C 180,E1 -19734.043,E2 -19734.043} C_VEL
LIN {X 0,Y 247.657,Z 458.141,A -85,B 0,C 180,E1 -19735.55,E2 -19735.55} C_VEL
LIN {X 0,Y 245.872,Z 447.33,A -85,B 0,C 180,E1 -19737.352,E2 -19737.352} C_VEL
LIN {X 0,Y 243.048,Z 436.083,A -85,B 0,C 180,E1 -19739.031,E2 -19739.031} C_VEL
LIN {X 0,Y 238.795,Z 423.82,A -85,B 0,C 180,E1 -19740.69,E2 -19740.69} C_VEL
LIN {X 0,Y 234.931,Z 414.644,A -85,B 0,C 180,E1 -19741.834,E2 -19741.834} C_VEL
LIN {X 0,Y 234.792,Z 413.959,A -85,B 0,C 180,E1 -19741.947,E2 -19741.947} C_VEL
LIN {X 0,Y 234.793,Z 411.412,A -85,B 0,C 180,E1 -19746.081,E2 -19746.081} C_VEL
LIN {X 0,Y 234.889,Z 411.227,A -85,B 0,C 180,E1 -19748.928,E2 -19748.928} C_VEL
LIN {X 0,Y 234.89,Z 411.225,A -85,B 0,C 180,E1 -19753.486,E2 -19753.486} C_VEL
LIN {X 0,Y 234.89,Z 411.228,A -85,B 0,C 180,E1 -19756.514,E2 -19756.514} C_VEL
LIN {X 0,Y 234.958,Z 411.213,A -85,B 0,C 180,E1 -19761.086,E2 -19761.086} C_VEL
LIN {X 0,Y 234.964,Z 411.213,A -85,B 0,C 180,E1 -19765.367,E2 -19765.367} C_VEL
LIN {X 0,Y 234.926,Z 411.221,A -85,B 0,C 180,E1 -19769.431,E2 -19769.431} C_VEL
LIN {X 0,Y 234.997,Z 411.213,A -85,B 0,C 180,E1 -19773.794,E2 -19773.794} C_VEL
LIN {X 0,Y 235.002,Z 411.211,A -85,B 0,C 180,E1 -19778.969,E2 -19778.969} C_VEL
LIN {X 0,Y 235.1,Z 411.198,A -85,B 0,C 180,E1 -19783.059,E2 -19783.059} C_VEL
LIN {X 0,Y 235.147,Z 411.196,A -85,B 0,C 180,E1 -19787.924,E2 -19787.924} C_VEL
LIN {X 0,Y 235.33,Z 411.172,A -85,B 0,C 180,E1 -19791.412,E2 -19791.412} C_VEL
LIN {X 0,Y 235.372,Z 411.165,A -85,B 0,C 180,E1 -19793.14,E2 -19793.14} C_VEL
LIN {X 0,Y 235.599,Z 411.139,A -85,B 0,C 180,E1 -19798.291,E2 -19798.291} C_VEL
LIN {X 0,Y 235.6,Z 411.141,A -85,B 0,C 180,E1 -19801.709,E2 -19801.709} C_VEL
LIN {X 0,Y 235.41,Z 411.161,A -85,B 0,C 180,E1 -19806.858,E2 -19806.858} C_VEL
LIN {X 0,Y 235.257,Z 411.181,A -85,B 0,C 180,E1 -19810.326,E2 -19810.326} C_VEL
